FUNCTION_BLOCK "LUps-M"   // FB1313, FBD
TITLE = LUps-M / LUps-M 2012-05-11
{ S7_Optimized_Access := 'FALSE' }
AUTHOR : VCC_JS
FAMILY : Actuator
NAME : LUps
VERSION : 0.2
// ================================================================================
// This module handles alarms from the UPS of type Murr electronic.
// When the conditions to generate the alarm disappear, a boolean output is 
// available to inform the upper level that the alarm can be reset.
// ================================================================================
// stored: AutoNumber false, IsIECCheckEnabled false, SetENOAutomatically False, UDAEnableTagReadback false
   VAR_INPUT
      I_UPSOk { ExternalAccessible := 'False'; ExternalVisible := 'False'; ExternalWritable := 'False'} : Bool;   // Input signal of UPS OK-signal
      I_SupplyVoltageOk { ExternalAccessible := 'False'; ExternalVisible := 'False'; ExternalWritable := 'False'} : Bool;   // Input signal supply voltage OK
      I_CapacitorOk { ExternalAccessible := 'False'; ExternalVisible := 'False'; ExternalWritable := 'False'} : Bool;   // Input signal Capacitor OK
      I_EnableAlarm { ExternalAccessible := 'False'; ExternalVisible := 'False'; ExternalWritable := 'False'} : Bool := TRUE;   // Enable alarm from upper level (0=disable/1=enable)
      I_AlarmResetPB { ExternalAccessible := 'False'; ExternalVisible := 'False'; ExternalWritable := 'False'} : Bool;   // Alarm reset pushbutton is activated
   END_VAR
   VAR_OUTPUT
      O_UPSOk { ExternalAccessible := 'False'; ExternalVisible := 'False'; ExternalWritable := 'False'} : Bool;   // UPS ok
      O_AlarmA { ExternalAccessible := 'False'; ExternalVisible := 'False'; ExternalWritable := 'False'} : Bool;   // Summation Alarm A.
      O_AlarmB { ExternalAccessible := 'False'; ExternalVisible := 'False'; ExternalWritable := 'False'} : Bool;   // Summation Alarm B.
      O_AlarmC { ExternalAccessible := 'False'; ExternalVisible := 'False'; ExternalWritable := 'False'} : Bool;   // Summation Alarm C.
      O_AlarmD { ExternalAccessible := 'False'; ExternalVisible := 'False'; ExternalWritable := 'False'} : Bool;   // Summation Alarm D.
      O_AlarmABCondition { ExternalAccessible := 'False'; ExternalVisible := 'False'; ExternalWritable := 'False'} : Bool;   // Alarm AB Condition
      H_IAnim { ExternalAccessible := 'False'; ExternalVisible := 'False'; ExternalWritable := 'False'} : Word;   // Icon animation
      H_AlarmWord { ExternalAccessible := 'False'; ExternalVisible := 'False'; ExternalWritable := 'False'} : DWord;   // Alarm Word
   END_VAR
   VAR DB_SPECIFIC
      AA_UPSFault { ExternalAccessible := 'False'; ExternalVisible := 'False'; ExternalWritable := 'False'} : Bool;   // UPS Fault / 0000: UPS Fault
      AD_SupplyVoltageAlarm { ExternalAccessible := 'False'; ExternalVisible := 'False'; ExternalWritable := 'False'} : Bool;   // Supply voltage not Ok / 0000: Supply voltage not Ok
      AD_UPSCapacitor { ExternalAccessible := 'False'; ExternalVisible := 'False'; ExternalWritable := 'False'} : Bool;   // UPS Capacitor warning / 0000: UPS Capacitor warning
      H_Out : Struct   // HMI
         Anim : Word;   // HMI Animation of the object
         DBnr : Int;   // HMI Animation DB number
      END_STRUCT;
      UPSCond { ExternalAccessible := 'False'; ExternalVisible := 'False'; ExternalWritable := 'False'} : Bool;   // Input condition to set the UPS alarm
      AlarmA { ExternalAccessible := 'False'; ExternalVisible := 'False'; ExternalWritable := 'False'} : Bool;   // Summation Alarm A
      AlarmB { ExternalAccessible := 'False'; ExternalVisible := 'False'; ExternalWritable := 'False'} : Bool;   // Summation Alarm B
      AlarmC { ExternalAccessible := 'False'; ExternalVisible := 'False'; ExternalWritable := 'False'} : Bool;   // Summation Alarm C
      AlarmD { ExternalAccessible := 'False'; ExternalVisible := 'False'; ExternalWritable := 'False'} : Bool;   // Summation Alarm D
      UPSOk { ExternalAccessible := 'False'; ExternalVisible := 'False'; ExternalWritable := 'False'} : Bool;   // UPS is ok
      DBnr { ExternalAccessible := 'False'; ExternalVisible := 'False'; ExternalWritable := 'False'} : Int;   // DB number
   END_VAR
BEGIN

NETWORK
TITLE = **** 1 - Inputs **** DB number
// DB number
      L     DINO;
      T     #DBnr;

REGION Network 2: **** 1 - Inputs **** The UPS alarm is active / **** 1 - Inputs ****
   // The UPS alarm is active
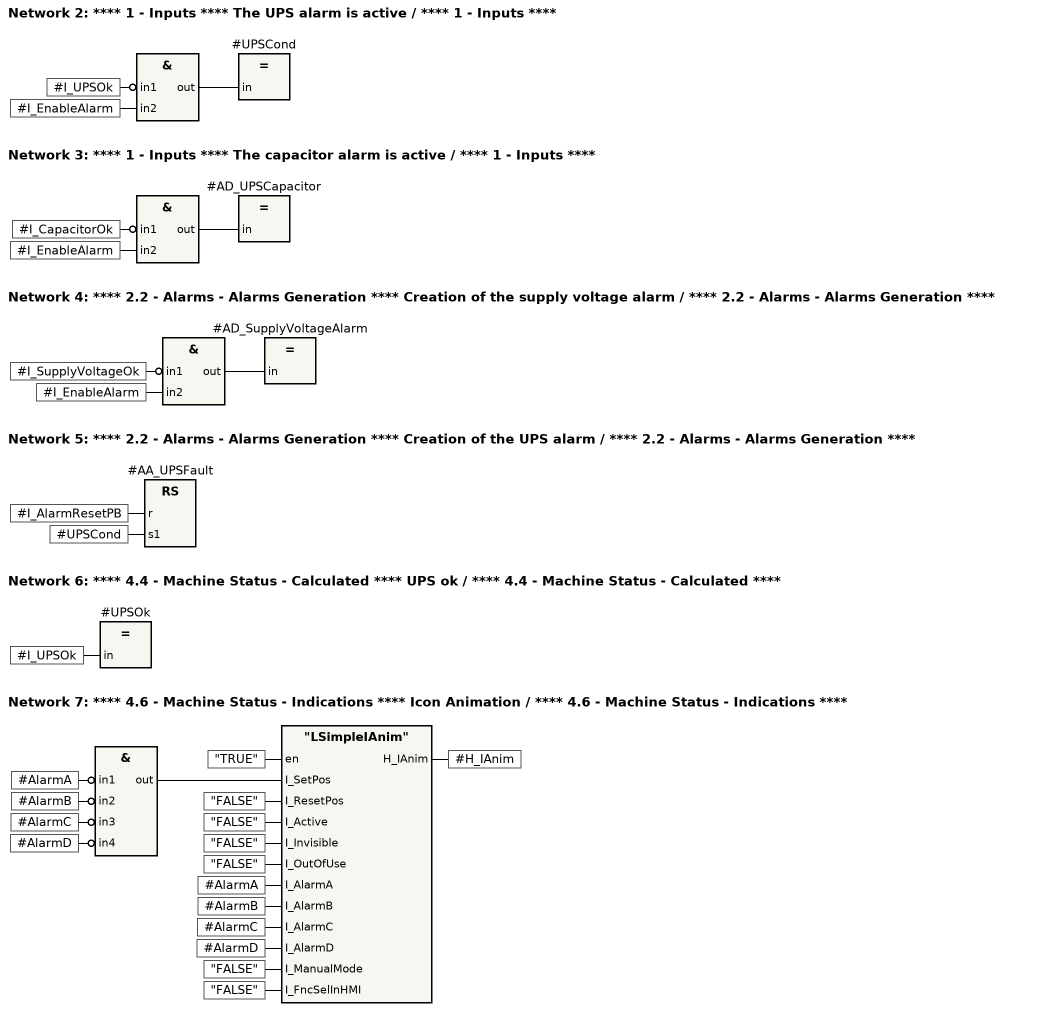
   #UPSCond := NOT #I_UPSOk AND #I_EnableAlarm;
END_REGION

REGION Network 3: **** 1 - Inputs **** The capacitor alarm is active / **** 1 - Inputs ****
   // The capacitor alarm is active
   #AD_UPSCapacitor := NOT #I_CapacitorOk AND #I_EnableAlarm;
END_REGION

REGION Network 4: **** 2.2 - Alarms - Alarms Generation **** Creation of the supply voltage alarm / **** 2.2 - Alarms - Alarms Generation ****
   // Creation of the supply voltage alarm
   #AD_SupplyVoltageAlarm := NOT #I_SupplyVoltageOk AND #I_EnableAlarm;
END_REGION

REGION Network 5: **** 2.2 - Alarms - Alarms Generation **** Creation of the UPS alarm / **** 2.2 - Alarms - Alarms Generation ****
   // Creation of the UPS alarm
   IF #I_AlarmResetPB THEN
       #AA_UPSFault := FALSE;   // RS flip-flop
   END_IF;
   IF #UPSCond THEN #AA_UPSFault := TRUE; END_IF;
END_REGION

REGION Network 6: **** 4.4 - Machine Status - Calculated **** UPS ok / **** 4.4 - Machine Status - Calculated ****
   // UPS ok
   #UPSOk := #I_UPSOk;
END_REGION

REGION Network 7: **** 4.6 - Machine Status - Indications **** Icon Animation / **** 4.6 - Machine Status - Indications ****
   // Icon Animation
   IF "TRUE" THEN
       "LSimpleIAnim"(I_SetPos := NOT #AlarmA AND NOT #AlarmB AND NOT #AlarmC AND NOT #AlarmD,
                      I_ResetPos := "FALSE",
                      I_Active := "FALSE",
                      I_Invisible := "FALSE",
                      I_OutOfUse := "FALSE",
                      I_AlarmA := #AlarmA,
                      I_AlarmB := #AlarmB,
                      I_AlarmC := #AlarmC,
                      I_AlarmD := #AlarmD,
                      I_ManualMode := "FALSE",
                      I_FncSelInHMI := "FALSE",
                      H_IAnim => #H_IAnim);
   END_IF;
END_REGION

REGION Network 8: **** 4.6 - Machine Status - Indications **** Animation / **** 4.6 - Machine Status - Indications ****
   // Animation
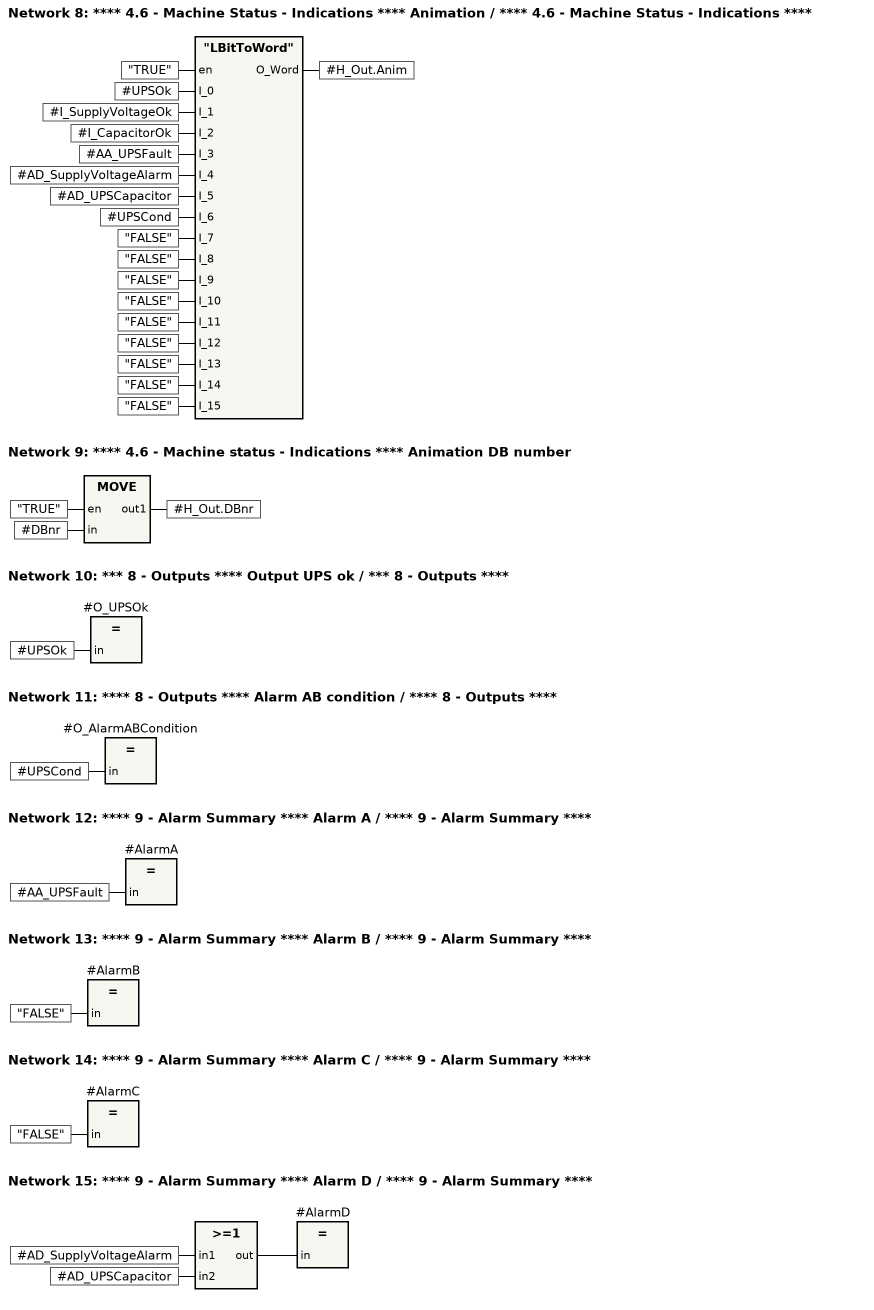
   IF "TRUE" THEN
       "LBitToWord"(I_0 := #UPSOk,
                    I_1 := #I_SupplyVoltageOk,
                    I_2 := #I_CapacitorOk,
                    I_3 := #AA_UPSFault,
                    I_4 := #AD_SupplyVoltageAlarm,
                    I_5 := #AD_UPSCapacitor,
                    I_6 := #UPSCond,
                    I_7 := "FALSE",
                    I_8 := "FALSE",
                    I_9 := "FALSE",
                    I_10 := "FALSE",
                    I_11 := "FALSE",
                    I_12 := "FALSE",
                    I_13 := "FALSE",
                    I_14 := "FALSE",
                    I_15 := "FALSE",
                    O_Word => #H_Out.Anim);
   END_IF;
END_REGION

REGION Network 9: **** 4.6 - Machine status - Indications **** Animation DB number
   // Animation DB number
   IF "TRUE" THEN #H_Out.DBnr := #DBnr; END_IF;
END_REGION

REGION Network 10: *** 8 - Outputs **** Output UPS ok / *** 8 - Outputs ****
   // Output UPS ok
   #O_UPSOk := #UPSOk;
END_REGION

REGION Network 11: **** 8 - Outputs **** Alarm AB condition / **** 8 - Outputs ****
   // Alarm AB Condition
   #O_AlarmABCondition := #UPSCond;
END_REGION

REGION Network 12: **** 9 - Alarm Summary **** Alarm A / **** 9 - Alarm Summary ****
   // Summary of alarms A
   #AlarmA := #AA_UPSFault;
END_REGION

REGION Network 13: **** 9 - Alarm Summary **** Alarm B / **** 9 - Alarm Summary ****
   // Summary of alarms B
   #AlarmB := "FALSE";
END_REGION

REGION Network 14: **** 9 - Alarm Summary **** Alarm C / **** 9 - Alarm Summary ****
   // Summary of alarms C
   #AlarmC := "FALSE";
END_REGION

REGION Network 15: **** 9 - Alarm Summary **** Alarm D / **** 9 - Alarm Summary ****
   // Summary of alarms D
   #AlarmD := #AD_SupplyVoltageAlarm OR #AD_UPSCapacitor;
END_REGION

REGION Network 16: **** 9.1 - Alarm Output **** Alarm A / **** 9 - Alarm Summary ****
   // Output of alarms A
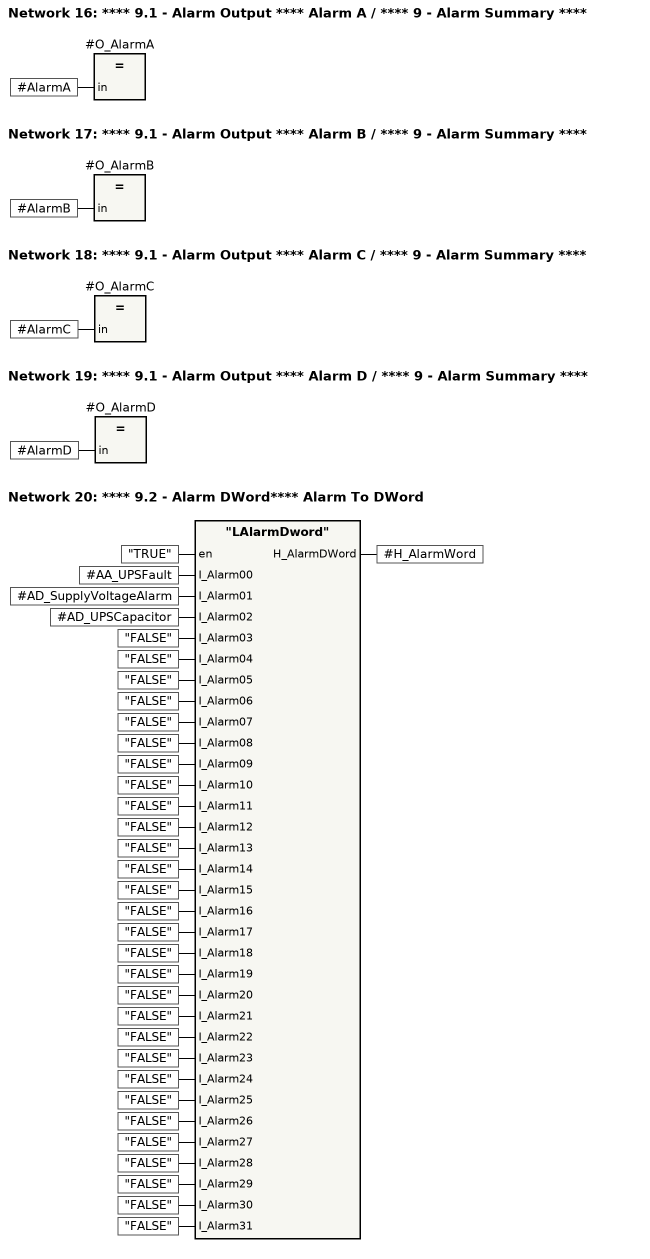
   #O_AlarmA := #AlarmA;
END_REGION

REGION Network 17: **** 9.1 - Alarm Output **** Alarm B / **** 9 - Alarm Summary ****
   // Output of alarms B
   #O_AlarmB := #AlarmB;
END_REGION

REGION Network 18: **** 9.1 - Alarm Output **** Alarm C / **** 9 - Alarm Summary ****
   // Output of alarms C
   #O_AlarmC := #AlarmC;
END_REGION

REGION Network 19: **** 9.1 - Alarm Output **** Alarm D / **** 9 - Alarm Summary ****
   // Output of alarms D
   #O_AlarmD := #AlarmD;
END_REGION

REGION Network 20: **** 9.2 - Alarm DWord**** Alarm To DWord
   // Alarm Word
   IF "TRUE" THEN
       "LAlarmDword"(I_Alarm00 := #AA_UPSFault,
                     I_Alarm01 := #AD_SupplyVoltageAlarm,
                     I_Alarm02 := #AD_UPSCapacitor,
                     I_Alarm03 := "FALSE",
                     I_Alarm04 := "FALSE",
                     I_Alarm05 := "FALSE",
                     I_Alarm06 := "FALSE",
                     I_Alarm07 := "FALSE",
                     I_Alarm08 := "FALSE",
                     I_Alarm09 := "FALSE",
                     I_Alarm10 := "FALSE",
                     I_Alarm11 := "FALSE",
                     I_Alarm12 := "FALSE",
                     I_Alarm13 := "FALSE",
                     I_Alarm14 := "FALSE",
                     I_Alarm15 := "FALSE",
                     I_Alarm16 := "FALSE",
                     I_Alarm17 := "FALSE",
                     I_Alarm18 := "FALSE",
                     I_Alarm19 := "FALSE",
                     I_Alarm20 := "FALSE",
                     I_Alarm21 := "FALSE",
                     I_Alarm22 := "FALSE",
                     I_Alarm23 := "FALSE",
                     I_Alarm24 := "FALSE",
                     I_Alarm25 := "FALSE",
                     I_Alarm26 := "FALSE",
                     I_Alarm27 := "FALSE",
                     I_Alarm28 := "FALSE",
                     I_Alarm29 := "FALSE",
                     I_Alarm30 := "FALSE",
                     I_Alarm31 := "FALSE",
                     H_AlarmDWord => #H_AlarmWord);
   END_IF;
END_REGION
END_FUNCTION_BLOCK

FUNCTION_BLOCK "LUps-Puls"   // FB1314, FBD
TITLE = LUps-M / LUps-M 2012-05-11 / LUps-Puls 2020-07-17
{ S7_Optimized_Access := 'FALSE' }
AUTHOR : VCC_JS
FAMILY : Actuator
NAME : LUps
VERSION : 0.2
// ================================================================================
// This module handles alarms from the UPS of type Murr electronic.
// When the conditions to generate the alarm disappear, a boolean output is 
// available to inform the upper level that the alarm can be reset.
// ================================================================================
// stored: AutoNumber false, IsIECCheckEnabled false, SetENOAutomatically False, UDAEnableTagReadback false
   VAR_INPUT
      I_Active { ExternalAccessible := 'False'; ExternalVisible := 'False'; ExternalWritable := 'False'} : Bool;   // Input signal of UPS Active-Signal / Input signal of UPS OK-signal
      I_Ready { ExternalAccessible := 'False'; ExternalVisible := 'False'; ExternalWritable := 'False'} : Bool;   // Input signal UPS Ready-Signal / Input signal supply voltage OK
      I_EnableAlarm { ExternalAccessible := 'False'; ExternalVisible := 'False'; ExternalWritable := 'False'} : Bool := TRUE;   // Enable alarm from upper level (0=disable/1=enable)
      I_AlarmResetPB { ExternalAccessible := 'False'; ExternalVisible := 'False'; ExternalWritable := 'False'} : Bool;   // Alarm reset pushbutton is activated
   END_VAR
   VAR_OUTPUT
      O_Active { ExternalAccessible := 'False'; ExternalVisible := 'False'; ExternalWritable := 'False'} : Bool;   // UPS Active / UPS ok
      O_AlarmA { ExternalAccessible := 'False'; ExternalVisible := 'False'; ExternalWritable := 'False'} : Bool;   // Summation Alarm A.
      O_AlarmB { ExternalAccessible := 'False'; ExternalVisible := 'False'; ExternalWritable := 'False'} : Bool;   // Summation Alarm B.
      O_AlarmC { ExternalAccessible := 'False'; ExternalVisible := 'False'; ExternalWritable := 'False'} : Bool;   // Summation Alarm C.
      O_AlarmD { ExternalAccessible := 'False'; ExternalVisible := 'False'; ExternalWritable := 'False'} : Bool;   // Summation Alarm D.
      O_AlarmABCondition { ExternalAccessible := 'False'; ExternalVisible := 'False'; ExternalWritable := 'False'} : Bool;   // Alarm AB Condition
      H_IAnim { ExternalAccessible := 'False'; ExternalVisible := 'False'; ExternalWritable := 'False'} : DWord;   // Icon animation
      H_AlarmWord { ExternalAccessible := 'False'; ExternalVisible := 'False'; ExternalWritable := 'False'} : DWord;   // Alarm Word
   END_VAR
   VAR DB_SPECIFIC
      AA_Active { ExternalAccessible := 'False'; ExternalVisible := 'False'; ExternalWritable := 'False'} : Bool;   // UPS Capaciter discharged / UPS Fault / 0000: UPS Fault
      AD_Ready { ExternalAccessible := 'False'; ExternalVisible := 'False'; ExternalWritable := 'False'} : Bool;   // UPS Ready-Signal / Supply voltage not Ok / 0000: Supply voltage not Ok
      H_Out : Struct   // HMI
         Anim : Word;   // HMI Animation of the object
         DBnr : Int;   // HMI Animation DB number
      END_STRUCT;
      UPSActiveAlarmCond { ExternalAccessible := 'False'; ExternalVisible := 'False'; ExternalWritable := 'False'} : Bool;   // Active condition to set the UPS alarm / Input condition to set the UPS alarm
      AlarmA { ExternalAccessible := 'False'; ExternalVisible := 'False'; ExternalWritable := 'False'} : Bool;   // Summation Alarm A
      AlarmB { ExternalAccessible := 'False'; ExternalVisible := 'False'; ExternalWritable := 'False'} : Bool;   // Summation Alarm B
      AlarmC { ExternalAccessible := 'False'; ExternalVisible := 'False'; ExternalWritable := 'False'} : Bool;   // Summation Alarm C
      AlarmD { ExternalAccessible := 'False'; ExternalVisible := 'False'; ExternalWritable := 'False'} : Bool;   // Summation Alarm D
      DBnr { ExternalAccessible := 'False'; ExternalVisible := 'False'; ExternalWritable := 'False'} : Int;   // DB number
   END_VAR
BEGIN

NETWORK
TITLE = **** 1 - Inputs **** DB number
// DB number
      L     DINO;
      T     #DBnr;

REGION Network 2: **** 1 - Inputs **** The UPS alarm is active / **** 1 - Inputs **** / **** 2.2 - Alarms - Alarms Generation **** UPS Not Active alarm condition
   // The UPS alarm is active / UPS Active alarm condition (Capacitors are  being discharged)
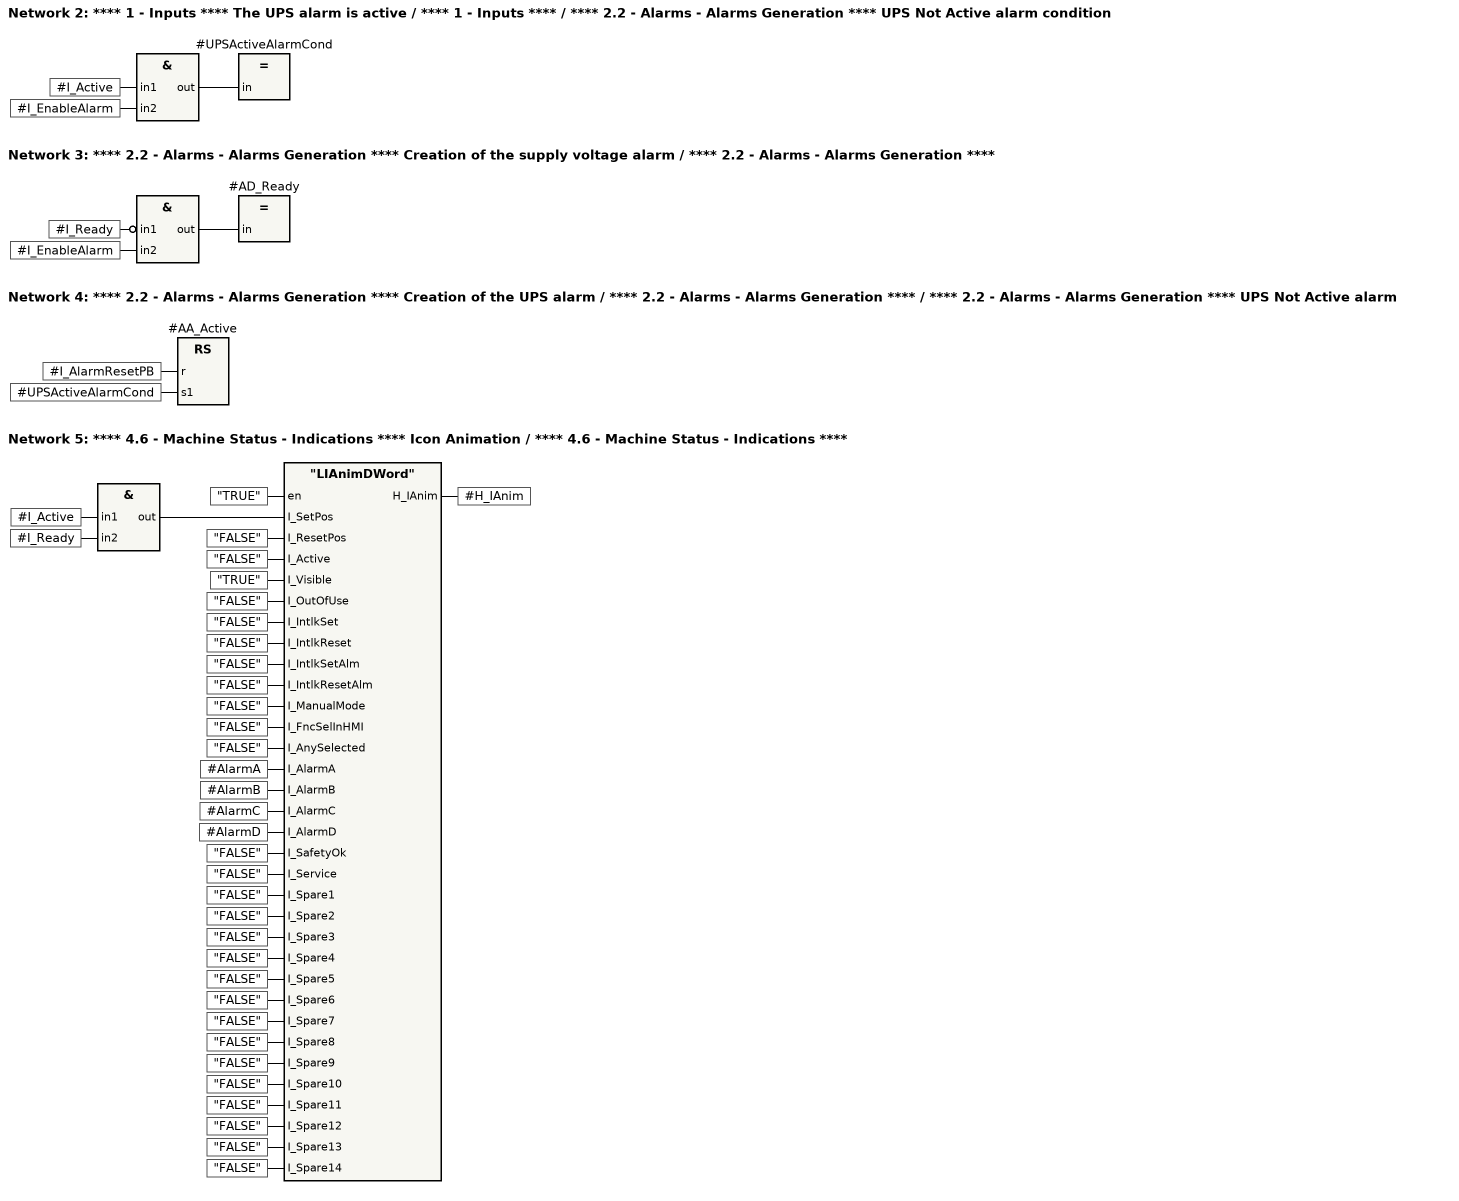
   #UPSActiveAlarmCond := #I_Active AND #I_EnableAlarm;
END_REGION

REGION Network 3: **** 2.2 - Alarms - Alarms Generation **** Creation of the supply voltage alarm / **** 2.2 - Alarms - Alarms Generation ****
   // Creation of the supply voltage alarm
   #AD_Ready := NOT #I_Ready AND #I_EnableAlarm;
END_REGION

REGION Network 4: **** 2.2 - Alarms - Alarms Generation **** Creation of the UPS alarm / **** 2.2 - Alarms - Alarms Generation **** / **** 2.2 - Alarms - Alarms Generation **** UPS Not Active alarm
   // Creation of the UPS alarm
   IF #I_AlarmResetPB THEN
       #AA_Active := FALSE;   // RS flip-flop
   END_IF;
   IF #UPSActiveAlarmCond THEN #AA_Active := TRUE; END_IF;
END_REGION

REGION Network 5: **** 4.6 - Machine Status - Indications **** Icon Animation / **** 4.6 - Machine Status - Indications ****
   // Icon Animation
   IF "TRUE" THEN
       "LIAnimDWord"(I_SetPos := #I_Active AND #I_Ready,
                     I_ResetPos := "FALSE",
                     I_Active := "FALSE",
                     I_Visible := "TRUE",
                     I_OutOfUse := "FALSE",
                     I_IntlkSet := "FALSE",
                     I_IntlkReset := "FALSE",
                     I_IntlkSetAlm := "FALSE",
                     I_IntlkResetAlm := "FALSE",
                     I_ManualMode := "FALSE",
                     I_FncSelInHMI := "FALSE",
                     I_AnySelected := "FALSE",
                     I_AlarmA := #AlarmA,
                     I_AlarmB := #AlarmB,
                     I_AlarmC := #AlarmC,
                     I_AlarmD := #AlarmD,
                     I_SafetyOk := "FALSE",
                     I_Service := "FALSE",
                     I_Spare1 := "FALSE",
                     I_Spare2 := "FALSE",
                     I_Spare3 := "FALSE",
                     I_Spare4 := "FALSE",
                     I_Spare5 := "FALSE",
                     I_Spare6 := "FALSE",
                     I_Spare7 := "FALSE",
                     I_Spare8 := "FALSE",
                     I_Spare9 := "FALSE",
                     I_Spare10 := "FALSE",
                     I_Spare11 := "FALSE",
                     I_Spare12 := "FALSE",
                     I_Spare13 := "FALSE",
                     I_Spare14 := "FALSE",
                     H_IAnim => #H_IAnim);
   END_IF;
END_REGION

REGION Network 6: **** 4.6 - Machine Status - Indications **** Animation / **** 4.6 - Machine Status - Indications ****
   // Animation
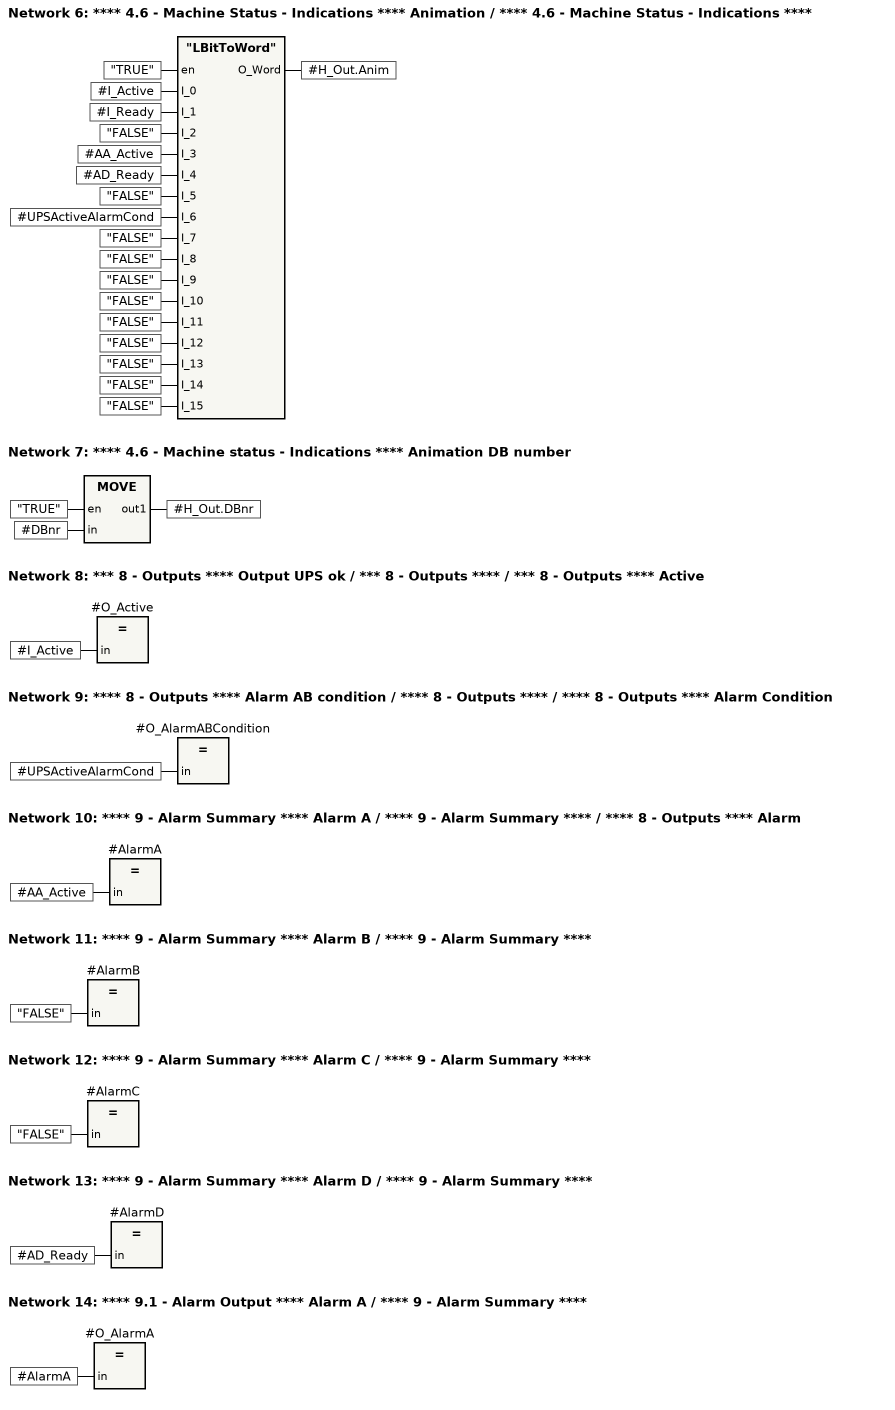
   IF "TRUE" THEN
       "LBitToWord"(I_0 := #I_Active,
                    I_1 := #I_Ready,
                    I_2 := "FALSE",
                    I_3 := #AA_Active,
                    I_4 := #AD_Ready,
                    I_5 := "FALSE",
                    I_6 := #UPSActiveAlarmCond,
                    I_7 := "FALSE",
                    I_8 := "FALSE",
                    I_9 := "FALSE",
                    I_10 := "FALSE",
                    I_11 := "FALSE",
                    I_12 := "FALSE",
                    I_13 := "FALSE",
                    I_14 := "FALSE",
                    I_15 := "FALSE",
                    O_Word => #H_Out.Anim);
   END_IF;
END_REGION

REGION Network 7: **** 4.6 - Machine status - Indications **** Animation DB number
   // Animation DB number
   IF "TRUE" THEN #H_Out.DBnr := #DBnr; END_IF;
END_REGION

REGION Network 8: *** 8 - Outputs **** Output UPS ok / *** 8 - Outputs **** / *** 8 - Outputs **** Active
   // Output UPS ok
   #O_Active := #I_Active;
END_REGION

REGION Network 9: **** 8 - Outputs **** Alarm AB condition / **** 8 - Outputs **** / **** 8 - Outputs **** Alarm Condition
   // Alarm AB Condition
   #O_AlarmABCondition := #UPSActiveAlarmCond;
END_REGION

REGION Network 10: **** 9 - Alarm Summary **** Alarm A / **** 9 - Alarm Summary **** / **** 8 - Outputs **** Alarm
   // Summary of alarms A / Alarm
   #AlarmA := #AA_Active;
END_REGION

REGION Network 11: **** 9 - Alarm Summary **** Alarm B / **** 9 - Alarm Summary ****
   // Summary of alarms B
   #AlarmB := "FALSE";
END_REGION

REGION Network 12: **** 9 - Alarm Summary **** Alarm C / **** 9 - Alarm Summary ****
   // Summary of alarms C
   #AlarmC := "FALSE";
END_REGION

REGION Network 13: **** 9 - Alarm Summary **** Alarm D / **** 9 - Alarm Summary ****
   // Summary of alarms D
   #AlarmD := #AD_Ready;
END_REGION

REGION Network 14: **** 9.1 - Alarm Output **** Alarm A / **** 9 - Alarm Summary ****
   // Output of alarms A
   #O_AlarmA := #AlarmA;
END_REGION

REGION Network 15: **** 9.1 - Alarm Output **** Alarm B / **** 9 - Alarm Summary ****
   // Output of alarms B
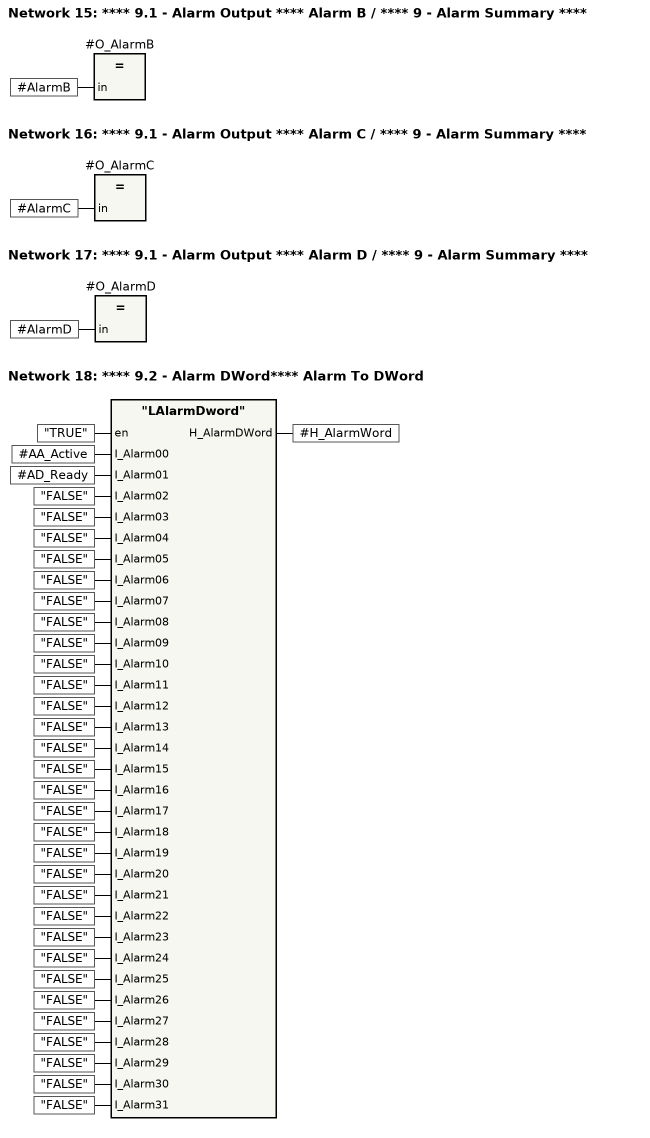
   #O_AlarmB := #AlarmB;
END_REGION

REGION Network 16: **** 9.1 - Alarm Output **** Alarm C / **** 9 - Alarm Summary ****
   // Output of alarms C
   #O_AlarmC := #AlarmC;
END_REGION

REGION Network 17: **** 9.1 - Alarm Output **** Alarm D / **** 9 - Alarm Summary ****
   // Output of alarms D
   #O_AlarmD := #AlarmD;
END_REGION

REGION Network 18: **** 9.2 - Alarm DWord**** Alarm To DWord
   // Alarm Word
   IF "TRUE" THEN
       "LAlarmDword"(I_Alarm00 := #AA_Active,
                     I_Alarm01 := #AD_Ready,
                     I_Alarm02 := "FALSE",
                     I_Alarm03 := "FALSE",
                     I_Alarm04 := "FALSE",
                     I_Alarm05 := "FALSE",
                     I_Alarm06 := "FALSE",
                     I_Alarm07 := "FALSE",
                     I_Alarm08 := "FALSE",
                     I_Alarm09 := "FALSE",
                     I_Alarm10 := "FALSE",
                     I_Alarm11 := "FALSE",
                     I_Alarm12 := "FALSE",
                     I_Alarm13 := "FALSE",
                     I_Alarm14 := "FALSE",
                     I_Alarm15 := "FALSE",
                     I_Alarm16 := "FALSE",
                     I_Alarm17 := "FALSE",
                     I_Alarm18 := "FALSE",
                     I_Alarm19 := "FALSE",
                     I_Alarm20 := "FALSE",
                     I_Alarm21 := "FALSE",
                     I_Alarm22 := "FALSE",
                     I_Alarm23 := "FALSE",
                     I_Alarm24 := "FALSE",
                     I_Alarm25 := "FALSE",
                     I_Alarm26 := "FALSE",
                     I_Alarm27 := "FALSE",
                     I_Alarm28 := "FALSE",
                     I_Alarm29 := "FALSE",
                     I_Alarm30 := "FALSE",
                     I_Alarm31 := "FALSE",
                     H_AlarmDWord => #H_AlarmWord);
   END_IF;
END_REGION
END_FUNCTION_BLOCK

FUNCTION_BLOCK "L1Alarm"   // FB1401, FBD
TITLE = L1Alarm / LProc1Alarm
{ S7_Optimized_Access := 'FALSE' }
AUTHOR : VCC
FAMILY : AlarmHnd
NAME : 1Alarm
VERSION : 1.0
// ================================================================================
// This module is used everywhere one alarm shall be generated when one (security) 
// input becomes True. The alarm have a delay time set in millieseconds.
// The alarm can be True only when the input Enable Alarm is also True.
// 
// When the conditions to generate the alarm is disappear, a boolean output is 
// available to inform the upper level that the alarm can be reset.
// The alarm is reset by means of the AlarmResetPB signal.
// ================================================================================
// stored: AutoNumber false, IsIECCheckEnabled false, SetENOAutomatically False, UDAEnableTagReadback false
   VAR_INPUT
      I_Input { ExternalAccessible := 'False'; ExternalVisible := 'False'; ExternalWritable := 'False'} : Bool;   // Input signal of the alarm
      I_AlarmClass { ExternalAccessible := 'False'; ExternalVisible := 'False'; ExternalWritable := 'False'} : Char;   // Alarm class -> A - B - C - D or E
      I_EnableAlarm { ExternalAccessible := 'False'; ExternalVisible := 'False'; ExternalWritable := 'False'} : Bool := TRUE;   // Enable alarm from upper level
      I_AlarmResetPB { ExternalAccessible := 'False'; ExternalVisible := 'False'; ExternalWritable := 'False'} : Bool;   // Alarm reset pushbutton is activated
      I_Invisible { ExternalAccessible := 'False'; ExternalVisible := 'False'; ExternalWritable := 'False'} : Bool;   // Invisible
      C_NcAlarm { ExternalAccessible := 'False'; ExternalVisible := 'False'; ExternalWritable := 'False'} : Bool;   // Alarm contact NC
   END_VAR
   VAR_OUTPUT
      O_Alarm { ExternalAccessible := 'False'; ExternalVisible := 'False'; ExternalWritable := 'False'} : Bool;   // Alarm
      O_AlarmABCondition { ExternalAccessible := 'False'; ExternalVisible := 'False'; ExternalWritable := 'False'} : Bool;   // Alarm AB condition
      H_IAnim { ExternalAccessible := 'False'; ExternalVisible := 'False'; ExternalWritable := 'False'} : Word;   // Icon animation
   END_VAR
   VAR DB_SPECIFIC
      H_Out : Struct   // HMI
         Anim : Word;   // HMI Animation of the object
         DBnr : Int;   // HMI Animation DB number
      END_STRUCT;
      Alarm { ExternalAccessible := 'False'; ExternalVisible := 'False'; ExternalWritable := 'False'} : Bool;   // Alarm
      AlarmClass_A { ExternalAccessible := 'False'; ExternalVisible := 'False'; ExternalWritable := 'False'} : Bool;   // The alarm is from alarm class A
      AlarmClass_B { ExternalAccessible := 'False'; ExternalVisible := 'False'; ExternalWritable := 'False'} : Bool;   // The alarm is from alarm class B
      AlarmClass_C { ExternalAccessible := 'False'; ExternalVisible := 'False'; ExternalWritable := 'False'} : Bool;   // The alarm is from alarm class C
      AlarmClass_D { ExternalAccessible := 'False'; ExternalVisible := 'False'; ExternalWritable := 'False'} : Bool;   // The alarm is from alarm class D
      AlarmClass_E { ExternalAccessible := 'False'; ExternalVisible := 'False'; ExternalWritable := 'False'} : Bool;   // The alarm is from alarm class E
      AlarmCond { ExternalAccessible := 'False'; ExternalVisible := 'False'; ExternalWritable := 'False'} : Bool;   // Alarm condition
      DBnr { ExternalAccessible := 'False'; ExternalVisible := 'False'; ExternalWritable := 'False'} : Int;   // HMI DB number
   END_VAR
BEGIN

NETWORK
TITLE = **** 1 - Inputs **** DB number
// DB number
      L     DINO;
      T     #DBnr;

NETWORK
TITLE = **** 1 - Inputs **** Alarm class
// Alarm class
// Alarm class = E
      L     #I_AlarmClass;
      L     'E';
      ==I;
      =     #AlarmClass_E;

// Alarm class = D
      L     #I_AlarmClass;
      L     'D';
      ==I;
      =     #AlarmClass_D;

// Alarm class = C
      L     #I_AlarmClass;
      L     'C';
      ==I;
      =     #AlarmClass_C;

// Alarm class = B
      L     #I_AlarmClass;
      L     'B';
      ==I;
      =     #AlarmClass_B;

// Alarm class = A
      AN    #AlarmClass_B;
      AN    #AlarmClass_C;
      AN    #AlarmClass_D;
      AN    #AlarmClass_E;
      =     #AlarmClass_A;


REGION Network 3: **** 2.2 - Alarms - Alarms Generation **** Alarm Condition
   // Condition for the Alarm
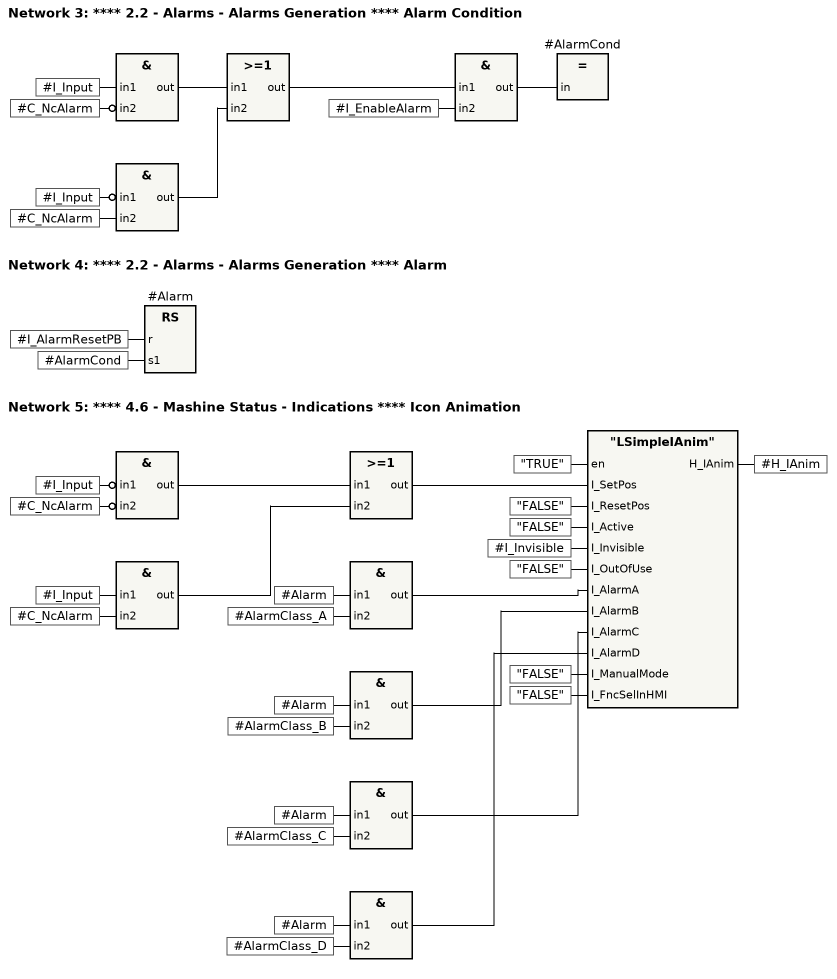
   #AlarmCond := ((#I_Input AND NOT #C_NcAlarm) OR (NOT #I_Input AND #C_NcAlarm)) AND #I_EnableAlarm;
END_REGION

REGION Network 4: **** 2.2 - Alarms - Alarms Generation **** Alarm
   // Creation of the Alarm
   IF #I_AlarmResetPB THEN
       #Alarm := FALSE;   // RS flip-flop
   END_IF;
   IF #AlarmCond THEN #Alarm := TRUE; END_IF;
END_REGION

REGION Network 5: **** 4.6 - Mashine Status - Indications **** Icon Animation
   // Icon Animation
   IF "TRUE" THEN
       "LSimpleIAnim"(I_SetPos := (NOT #I_Input AND NOT #C_NcAlarm) OR (#I_Input AND #C_NcAlarm),
                      I_ResetPos := "FALSE",
                      I_Active := "FALSE",
                      I_Invisible := #I_Invisible,
                      I_OutOfUse := "FALSE",
                      I_AlarmA := #Alarm AND #AlarmClass_A,
                      I_AlarmB := #Alarm AND #AlarmClass_B,
                      I_AlarmC := #Alarm AND #AlarmClass_C,
                      I_AlarmD := #Alarm AND #AlarmClass_D,
                      I_ManualMode := "FALSE",
                      I_FncSelInHMI := "FALSE",
                      H_IAnim => #H_IAnim);
   END_IF;
END_REGION

REGION Network 6: **** 4.6 - Machine Status - Indications **** Animation
   // Animation
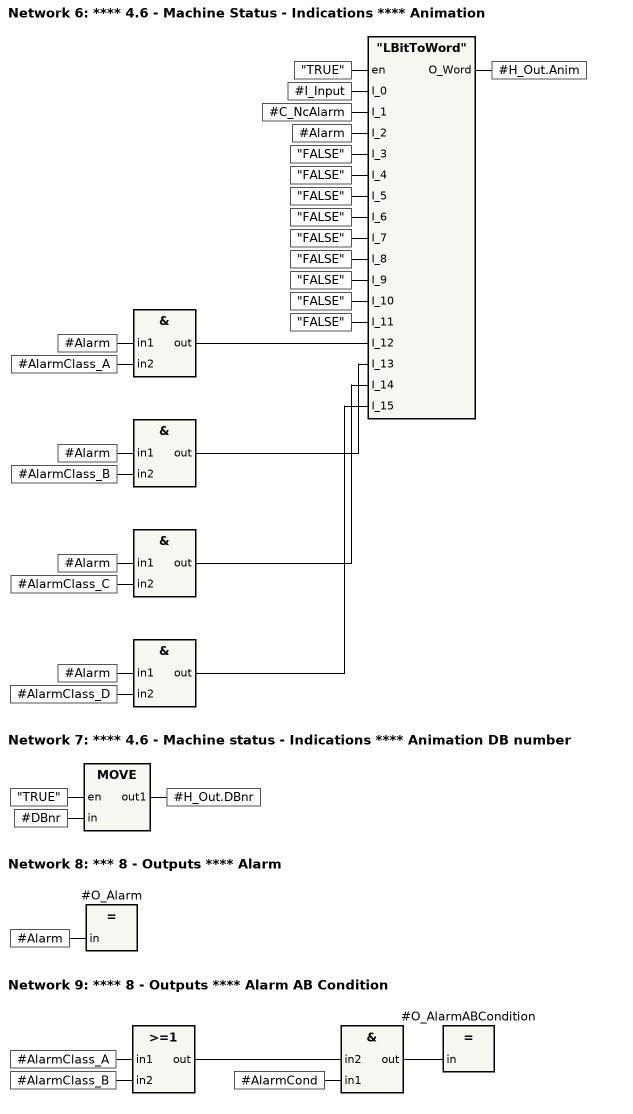
   IF "TRUE" THEN
       "LBitToWord"(I_0 := #I_Input,
                    I_1 := #C_NcAlarm,
                    I_2 := #Alarm,
                    I_3 := "FALSE",
                    I_4 := "FALSE",
                    I_5 := "FALSE",
                    I_6 := "FALSE",
                    I_7 := "FALSE",
                    I_8 := "FALSE",
                    I_9 := "FALSE",
                    I_10 := "FALSE",
                    I_11 := "FALSE",
                    I_12 := #Alarm AND #AlarmClass_A,
                    I_13 := #Alarm AND #AlarmClass_B,
                    I_14 := #Alarm AND #AlarmClass_C,
                    I_15 := #Alarm AND #AlarmClass_D,
                    O_Word => #H_Out.Anim);
   END_IF;
END_REGION

REGION Network 7: **** 4.6 - Machine status - Indications **** Animation DB number
   // Animation DB number
   IF "TRUE" THEN #H_Out.DBnr := #DBnr; END_IF;
END_REGION

REGION Network 8: *** 8 - Outputs **** Alarm
   // Output of the Alarm
   #O_Alarm := #Alarm;
END_REGION

REGION Network 9: **** 8 - Outputs **** Alarm AB Condition
   // Alarm Resetable
   #O_AlarmABCondition := (#AlarmClass_A OR #AlarmClass_B) AND #AlarmCond;
END_REGION
END_FUNCTION_BLOCK

FUNCTION_BLOCK "L5Alarm"   // FB1405, FBD
TITLE = L5Alarm
{ S7_Optimized_Access := 'FALSE' }
AUTHOR : VCC
FAMILY : AlarmHnd
NAME : 5Alarm
VERSION : 1.0
// ================================================================================
// This module is used everywhere 5 alarms has to be generated when one (security) 
// corresponding input becomes True.
// All alarms can be True only when the corresponding input Enable Alarm is also 
// True.
// When the conditions to generate the alarm is disappear, a boolean (one per 
// alarm) available to inform the upper level that the corresponding alarm can be 
// reset.
// All alarms are reset by means of the AlarmResetPB signal.
// ================================================================================
// stored: AutoNumber false, IsIECCheckEnabled false, SetENOAutomatically False, UDAEnableTagReadback false
   VAR_INPUT
      I_Input1 { ExternalAccessible := 'False'; ExternalVisible := 'False'; ExternalWritable := 'False'} : Bool;   // Input alarm 1
      I_AlarmClass1 { ExternalAccessible := 'False'; ExternalVisible := 'False'; ExternalWritable := 'False'} : Char;   // Alarm class -> A - B - C - D or E
      I_EnableAlarm1 { ExternalAccessible := 'False'; ExternalVisible := 'False'; ExternalWritable := 'False'} : Bool := TRUE;   // Enable alarm 1 from upper level
      I_Invisible1 { ExternalAccessible := 'False'; ExternalVisible := 'False'; ExternalWritable := 'False'} : Bool;   // Invisible 1
      I_Input2 { ExternalAccessible := 'False'; ExternalVisible := 'False'; ExternalWritable := 'False'} : Bool;   // Input alarm 2
      I_AlarmClass2 { ExternalAccessible := 'False'; ExternalVisible := 'False'; ExternalWritable := 'False'} : Char;   // Alarm class -> A - B - C - D or E
      I_EnableAlarm2 { ExternalAccessible := 'False'; ExternalVisible := 'False'; ExternalWritable := 'False'} : Bool := TRUE;   // Enable alarm 2 from upper level
      I_Invisible2 { ExternalAccessible := 'False'; ExternalVisible := 'False'; ExternalWritable := 'False'} : Bool;   // Invisible 2
      I_Input3 { ExternalAccessible := 'False'; ExternalVisible := 'False'; ExternalWritable := 'False'} : Bool;   // Input alarm 3
      I_AlarmClass3 { ExternalAccessible := 'False'; ExternalVisible := 'False'; ExternalWritable := 'False'} : Char;   // Alarm class -> A - B - C - D or E
      I_EnableAlarm3 { ExternalAccessible := 'False'; ExternalVisible := 'False'; ExternalWritable := 'False'} : Bool := TRUE;   // Enable alarm 3 from upper level
      I_Invisible3 { ExternalAccessible := 'False'; ExternalVisible := 'False'; ExternalWritable := 'False'} : Bool;   // Invisible 3
      I_Input4 { ExternalAccessible := 'False'; ExternalVisible := 'False'; ExternalWritable := 'False'} : Bool;   // Input alarm 4
      I_AlarmClass4 { ExternalAccessible := 'False'; ExternalVisible := 'False'; ExternalWritable := 'False'} : Char;   // Alarm class -> A - B - C - D or E
      I_EnableAlarm4 { ExternalAccessible := 'False'; ExternalVisible := 'False'; ExternalWritable := 'False'} : Bool := TRUE;   // Enable alarm 4 from upper level
      I_Invisible4 { ExternalAccessible := 'False'; ExternalVisible := 'False'; ExternalWritable := 'False'} : Bool;   // Invisible 4
      I_Input5 { ExternalAccessible := 'False'; ExternalVisible := 'False'; ExternalWritable := 'False'} : Bool;   // Input alarm 5
      I_AlarmClass5 { ExternalAccessible := 'False'; ExternalVisible := 'False'; ExternalWritable := 'False'} : Char;   // Alarm class -> A - B - C - D or E
      I_EnableAlarm5 { ExternalAccessible := 'False'; ExternalVisible := 'False'; ExternalWritable := 'False'} : Bool := TRUE;   // Enable alarm 5 from upper level
      I_Invisible5 { ExternalAccessible := 'False'; ExternalVisible := 'False'; ExternalWritable := 'False'} : Bool;   // Invisible
      I_AlarmResetPB { ExternalAccessible := 'False'; ExternalVisible := 'False'; ExternalWritable := 'False'} : Bool;   // Alarm reset pushbutton is activated
   END_VAR
   VAR_OUTPUT
      O_Alarm1 { ExternalAccessible := 'False'; ExternalVisible := 'False'; ExternalWritable := 'False'} : Bool;   // Alarm 1
      O_Alarm2 { ExternalAccessible := 'False'; ExternalVisible := 'False'; ExternalWritable := 'False'} : Bool;   // Alarm 2
      O_Alarm3 { ExternalAccessible := 'False'; ExternalVisible := 'False'; ExternalWritable := 'False'} : Bool;   // Alarm 3
      O_Alarm4 { ExternalAccessible := 'False'; ExternalVisible := 'False'; ExternalWritable := 'False'} : Bool;   // Alarm 4
      O_Alarm5 { ExternalAccessible := 'False'; ExternalVisible := 'False'; ExternalWritable := 'False'} : Bool;   // Alarm 5
      O_AlarmABCondition { ExternalAccessible := 'False'; ExternalVisible := 'False'; ExternalWritable := 'False'} : Bool;   // Alarm AB condition
      H_IAnim1 { ExternalAccessible := 'False'; ExternalVisible := 'False'; ExternalWritable := 'False'} : Word;   // Icon Animation 1
      H_IAnim2 { ExternalAccessible := 'False'; ExternalVisible := 'False'; ExternalWritable := 'False'} : Word;   // Icon Animation 2
      H_IAnim3 { ExternalAccessible := 'False'; ExternalVisible := 'False'; ExternalWritable := 'False'} : Word;   // Icon Animation 3
      H_IAnim4 { ExternalAccessible := 'False'; ExternalVisible := 'False'; ExternalWritable := 'False'} : Word;   // Icon Animation 4
      H_IAnim5 { ExternalAccessible := 'False'; ExternalVisible := 'False'; ExternalWritable := 'False'} : Word;   // Icon Animation 5
   END_VAR
   VAR DB_SPECIFIC
      H_Out : Struct   // HMI
         Anim1 : Word;   // HMI Animation of the object
         Anim2 : Word;   // HMI Animation of the object
         Anim3 : Word;   // HMI Animation of the object
         Anim4 : Word;   // HMI Animation of the object
         Anim5 : Word;   // HMI Animation of the object
         DBnr : Int;   // HMI Animation DB number
      END_STRUCT;
      Alarm1 { ExternalAccessible := 'False'; ExternalVisible := 'False'; ExternalWritable := 'False'} : Bool;   // Alarm 1
      AlarmClass1_A { ExternalAccessible := 'False'; ExternalVisible := 'False'; ExternalWritable := 'False'} : Bool;   // The alarm is from alarm class A
      AlarmClass1_B { ExternalAccessible := 'False'; ExternalVisible := 'False'; ExternalWritable := 'False'} : Bool;   // The alarm is from alarm class B
      AlarmClass1_C { ExternalAccessible := 'False'; ExternalVisible := 'False'; ExternalWritable := 'False'} : Bool;   // The alarm is from alarm class C
      AlarmClass1_D { ExternalAccessible := 'False'; ExternalVisible := 'False'; ExternalWritable := 'False'} : Bool;   // The alarm is from alarm class D
      AlarmClass1_E { ExternalAccessible := 'False'; ExternalVisible := 'False'; ExternalWritable := 'False'} : Bool;   // The alarm is from alarm class E
      Alarm1Cond { ExternalAccessible := 'False'; ExternalVisible := 'False'; ExternalWritable := 'False'} : Bool;   // Alarm 1 condition
      Alarm2 { ExternalAccessible := 'False'; ExternalVisible := 'False'; ExternalWritable := 'False'} : Bool;   // Alarm 2
      AlarmClass2_A { ExternalAccessible := 'False'; ExternalVisible := 'False'; ExternalWritable := 'False'} : Bool;   // The alarm is from alarm class A
      AlarmClass2_B { ExternalAccessible := 'False'; ExternalVisible := 'False'; ExternalWritable := 'False'} : Bool;   // The alarm is from alarm class B
      AlarmClass2_C { ExternalAccessible := 'False'; ExternalVisible := 'False'; ExternalWritable := 'False'} : Bool;   // The alarm is from alarm class C
      AlarmClass2_D { ExternalAccessible := 'False'; ExternalVisible := 'False'; ExternalWritable := 'False'} : Bool;   // The alarm is from alarm class D
      AlarmClass2_E { ExternalAccessible := 'False'; ExternalVisible := 'False'; ExternalWritable := 'False'} : Bool;   // The alarm is from alarm class E
      Alarm2Cond { ExternalAccessible := 'False'; ExternalVisible := 'False'; ExternalWritable := 'False'} : Bool;   // Alarm 2 condition
      Alarm3 { ExternalAccessible := 'False'; ExternalVisible := 'False'; ExternalWritable := 'False'} : Bool;   // Alarm 3
      AlarmClass3_A { ExternalAccessible := 'False'; ExternalVisible := 'False'; ExternalWritable := 'False'} : Bool;   // The alarm is from alarm class A
      AlarmClass3_B { ExternalAccessible := 'False'; ExternalVisible := 'False'; ExternalWritable := 'False'} : Bool;   // The alarm is from alarm class B
      AlarmClass3_C { ExternalAccessible := 'False'; ExternalVisible := 'False'; ExternalWritable := 'False'} : Bool;   // The alarm is from alarm class C
      AlarmClass3_D { ExternalAccessible := 'False'; ExternalVisible := 'False'; ExternalWritable := 'False'} : Bool;   // The alarm is from alarm class D
      AlarmClass3_E { ExternalAccessible := 'False'; ExternalVisible := 'False'; ExternalWritable := 'False'} : Bool;   // The alarm is from alarm class E
      Alarm3Cond { ExternalAccessible := 'False'; ExternalVisible := 'False'; ExternalWritable := 'False'} : Bool;   // Alarm 3 condition
      Alarm4 { ExternalAccessible := 'False'; ExternalVisible := 'False'; ExternalWritable := 'False'} : Bool;   // Alarm 4
      AlarmClass4_A { ExternalAccessible := 'False'; ExternalVisible := 'False'; ExternalWritable := 'False'} : Bool;   // The alarm is from alarm class A
      AlarmClass4_B { ExternalAccessible := 'False'; ExternalVisible := 'False'; ExternalWritable := 'False'} : Bool;   // The alarm is from alarm class B
      AlarmClass4_C { ExternalAccessible := 'False'; ExternalVisible := 'False'; ExternalWritable := 'False'} : Bool;   // The alarm is from alarm class C
      AlarmClass4_D { ExternalAccessible := 'False'; ExternalVisible := 'False'; ExternalWritable := 'False'} : Bool;   // The alarm is from alarm class D
      AlarmClass4_E { ExternalAccessible := 'False'; ExternalVisible := 'False'; ExternalWritable := 'False'} : Bool;   // The alarm is from alarm class E
      Alarm4Cond { ExternalAccessible := 'False'; ExternalVisible := 'False'; ExternalWritable := 'False'} : Bool;   // Alarm 4 condition
      Alarm5 { ExternalAccessible := 'False'; ExternalVisible := 'False'; ExternalWritable := 'False'} : Bool;   // Alarm 5
      AlarmClass5_A { ExternalAccessible := 'False'; ExternalVisible := 'False'; ExternalWritable := 'False'} : Bool;   // The alarm is from alarm class A
      AlarmClass5_B { ExternalAccessible := 'False'; ExternalVisible := 'False'; ExternalWritable := 'False'} : Bool;   // The alarm is from alarm class B
      AlarmClass5_C { ExternalAccessible := 'False'; ExternalVisible := 'False'; ExternalWritable := 'False'} : Bool;   // The alarm is from alarm class C
      AlarmClass5_D { ExternalAccessible := 'False'; ExternalVisible := 'False'; ExternalWritable := 'False'} : Bool;   // The alarm is from alarm class D
      AlarmClass5_E { ExternalAccessible := 'False'; ExternalVisible := 'False'; ExternalWritable := 'False'} : Bool;   // The alarm is from alarm class E
      Alarm5Cond { ExternalAccessible := 'False'; ExternalVisible := 'False'; ExternalWritable := 'False'} : Bool;   // Alarm 5 condition
      DBnr { ExternalAccessible := 'False'; ExternalVisible := 'False'; ExternalWritable := 'False'} : Int;   // HMI DB number
   END_VAR
BEGIN

NETWORK
TITLE = **** 1 - Inputs **** DB number
// DB number
      L     DINO;
      T     #DBnr;

NETWORK
TITLE = **** 1 - Inputs **** Alarm class 1
// Alarm class
// Alarm class = E
      L     #I_AlarmClass1;
      L     'E';
      ==I;
      =     #AlarmClass1_E;

// Alarm class = D
      L     #I_AlarmClass1;
      L     'D';
      ==I;
      =     #AlarmClass1_D;

// Alarm class = C
      L     #I_AlarmClass1;
      L     'C';
      ==I;
      =     #AlarmClass1_C;

// Alarm class = B
      L     #I_AlarmClass1;
      L     'B';
      ==I;
      =     #AlarmClass1_B;

// Alarm class = A
      AN    #AlarmClass1_B;
      AN    #AlarmClass1_C;
      AN    #AlarmClass1_D;
      AN    #AlarmClass1_E;
      =     #AlarmClass1_A;


NETWORK
TITLE = **** 1 - Inputs **** Alarm class 2
// Alarm class
// Alarm class = E
      L     #I_AlarmClass2;
      L     'E';
      ==I;
      =     #AlarmClass2_E;

// Alarm class = D
      L     #I_AlarmClass2;
      L     'D';
      ==I;
      =     #AlarmClass2_D;

// Alarm class = C
      L     #I_AlarmClass2;
      L     'C';
      ==I;
      =     #AlarmClass2_C;

// Alarm class = B
      L     #I_AlarmClass2;
      L     'B';
      ==I;
      =     #AlarmClass2_B;

// Alarm class = A
      AN    #AlarmClass2_B;
      AN    #AlarmClass2_C;
      AN    #AlarmClass2_D;
      AN    #AlarmClass2_E;
      =     #AlarmClass2_A;


NETWORK
TITLE = **** 1 - Inputs **** Alarm class 3
// Alarm class
// Alarm class = E
      L     #I_AlarmClass3;
      L     'E';
      ==I;
      =     #AlarmClass3_E;

// Alarm class = D
      L     #I_AlarmClass3;
      L     'D';
      ==I;
      =     #AlarmClass3_D;

// Alarm class = C
      L     #I_AlarmClass3;
      L     'C';
      ==I;
      =     #AlarmClass3_C;

// Alarm class = B
      L     #I_AlarmClass3;
      L     'B';
      ==I;
      =     #AlarmClass3_B;

// Alarm class = A
      AN    #AlarmClass3_B;
      AN    #AlarmClass3_C;
      AN    #AlarmClass3_D;
      AN    #AlarmClass3_E;
      =     #AlarmClass3_A;


NETWORK
TITLE = **** 1 - Inputs **** Alarm class 4
// Alarm class
// Alarm class = E
      L     #I_AlarmClass4;
      L     'E';
      ==I;
      =     #AlarmClass4_E;

// Alarm class = D
      L     #I_AlarmClass4;
      L     'D';
      ==I;
      =     #AlarmClass4_D;

// Alarm class = C
      L     #I_AlarmClass4;
      L     'C';
      ==I;
      =     #AlarmClass4_C;

// Alarm class = B
      L     #I_AlarmClass4;
      L     'B';
      ==I;
      =     #AlarmClass4_B;

// Alarm class = A
      AN    #AlarmClass4_B;
      AN    #AlarmClass4_C;
      AN    #AlarmClass4_D;
      AN    #AlarmClass4_E;
      =     #AlarmClass4_A;


NETWORK
TITLE = **** 1 - Inputs **** Alarm class 5
// Alarm class
// Alarm class = E
      L     #I_AlarmClass5;
      L     'E';
      ==I;
      =     #AlarmClass5_E;

// Alarm class = D
      L     #I_AlarmClass5;
      L     'D';
      ==I;
      =     #AlarmClass5_D;

// Alarm class = C
      L     #I_AlarmClass5;
      L     'C';
      ==I;
      =     #AlarmClass5_C;

// Alarm class = B
      L     #I_AlarmClass5;
      L     'B';
      ==I;
      =     #AlarmClass5_B;

// Alarm class = A
      AN    #AlarmClass5_B;
      AN    #AlarmClass5_C;
      AN    #AlarmClass5_D;
      AN    #AlarmClass5_E;
      =     #AlarmClass5_A;


REGION Network 7: **** 2.2 - Alarms - Alarms Generation **** Alarm Condition 1
   // Condition for Alarm 1
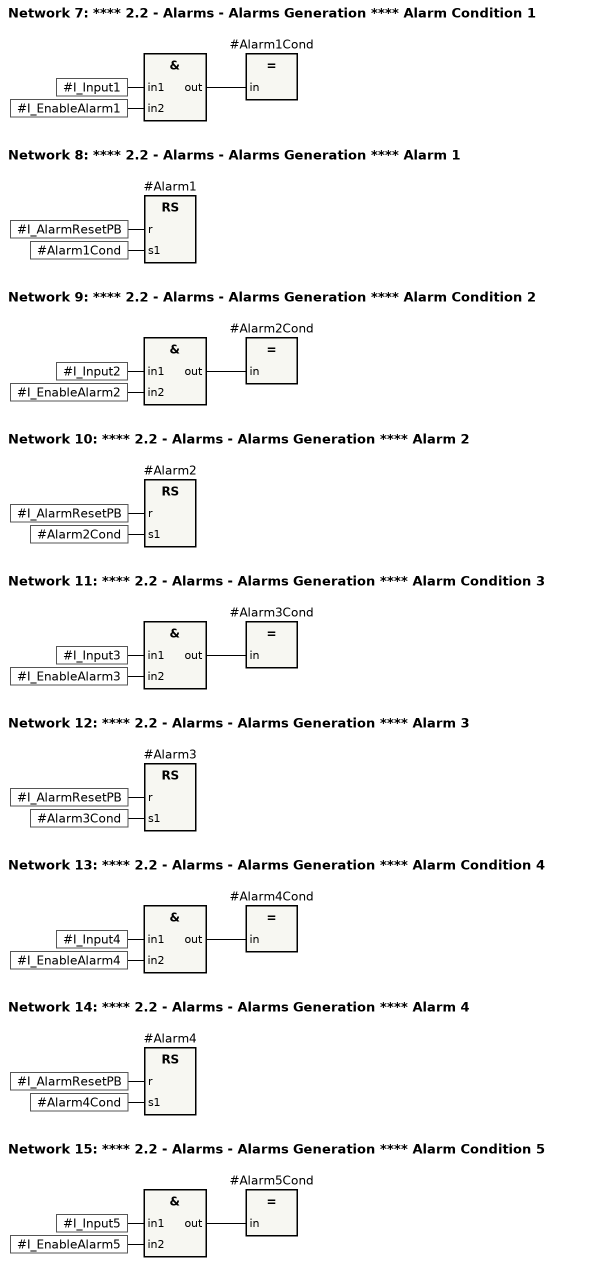
   #Alarm1Cond := #I_Input1 AND #I_EnableAlarm1;
END_REGION

REGION Network 8: **** 2.2 - Alarms - Alarms Generation **** Alarm 1
   // Creation of the Alarm 1
   IF #I_AlarmResetPB THEN
       #Alarm1 := FALSE;   // RS flip-flop
   END_IF;
   IF #Alarm1Cond THEN #Alarm1 := TRUE; END_IF;
END_REGION

REGION Network 9: **** 2.2 - Alarms - Alarms Generation **** Alarm Condition 2
   // Condition for Alarm 2
   #Alarm2Cond := #I_Input2 AND #I_EnableAlarm2;
END_REGION

REGION Network 10: **** 2.2 - Alarms - Alarms Generation **** Alarm 2
   // Creation of the Alarm 2
   IF #I_AlarmResetPB THEN
       #Alarm2 := FALSE;   // RS flip-flop
   END_IF;
   IF #Alarm2Cond THEN #Alarm2 := TRUE; END_IF;
END_REGION

REGION Network 11: **** 2.2 - Alarms - Alarms Generation **** Alarm Condition 3
   // Condition for Alarm 3
   #Alarm3Cond := #I_Input3 AND #I_EnableAlarm3;
END_REGION

REGION Network 12: **** 2.2 - Alarms - Alarms Generation **** Alarm 3
   // Creation of the Alarm 3
   IF #I_AlarmResetPB THEN
       #Alarm3 := FALSE;   // RS flip-flop
   END_IF;
   IF #Alarm3Cond THEN #Alarm3 := TRUE; END_IF;
END_REGION

REGION Network 13: **** 2.2 - Alarms - Alarms Generation **** Alarm Condition 4
   // Condition for Alarm 4
   #Alarm4Cond := #I_Input4 AND #I_EnableAlarm4;
END_REGION

REGION Network 14: **** 2.2 - Alarms - Alarms Generation **** Alarm 4
   // Creation of the Alarm 4
   IF #I_AlarmResetPB THEN
       #Alarm4 := FALSE;   // RS flip-flop
   END_IF;
   IF #Alarm4Cond THEN #Alarm4 := TRUE; END_IF;
END_REGION

REGION Network 15: **** 2.2 - Alarms - Alarms Generation **** Alarm Condition 5
   // Condition for Alarm 5
   #Alarm5Cond := #I_Input5 AND #I_EnableAlarm5;
END_REGION

REGION Network 16: **** 2.2 - Alarms - Alarms Generation **** Alarm 5
   // Creation of the Alarm 5
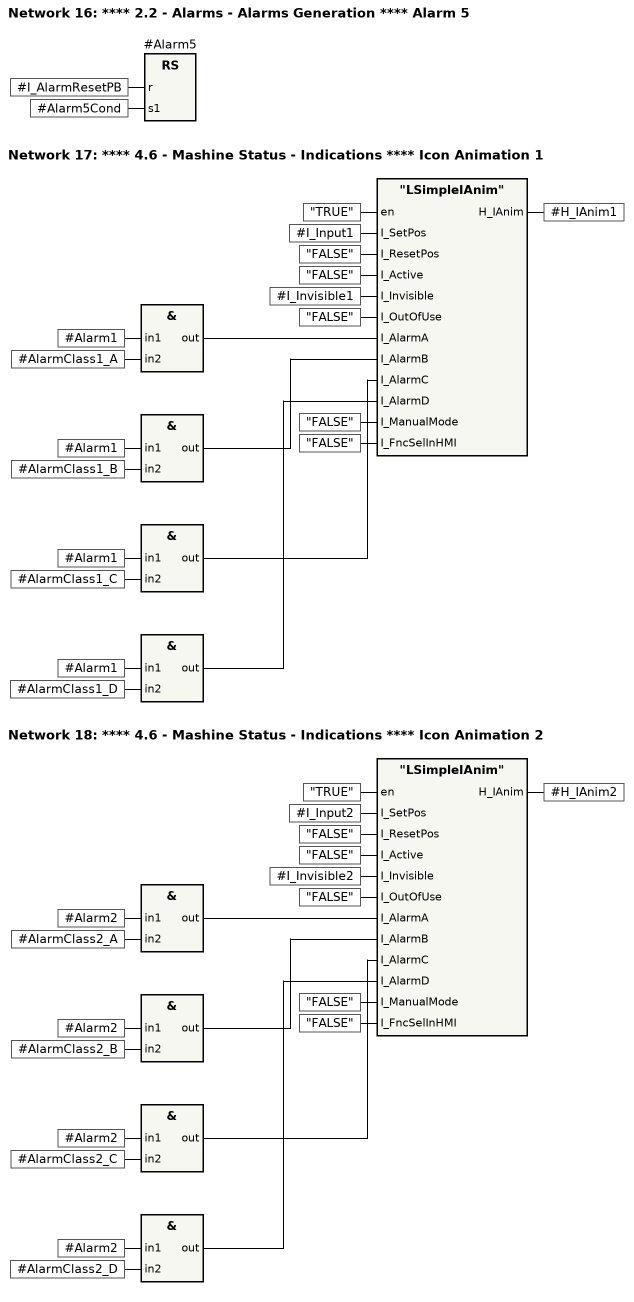
   IF #I_AlarmResetPB THEN
       #Alarm5 := FALSE;   // RS flip-flop
   END_IF;
   IF #Alarm5Cond THEN #Alarm5 := TRUE; END_IF;
END_REGION

REGION Network 17: **** 4.6 - Mashine Status - Indications **** Icon Animation 1
   // Icon Animation 1
   IF "TRUE" THEN
       "LSimpleIAnim"(I_SetPos := #I_Input1,
                      I_ResetPos := "FALSE",
                      I_Active := "FALSE",
                      I_Invisible := #I_Invisible1,
                      I_OutOfUse := "FALSE",
                      I_AlarmA := #Alarm1 AND #AlarmClass1_A,
                      I_AlarmB := #Alarm1 AND #AlarmClass1_B,
                      I_AlarmC := #Alarm1 AND #AlarmClass1_C,
                      I_AlarmD := #Alarm1 AND #AlarmClass1_D,
                      I_ManualMode := "FALSE",
                      I_FncSelInHMI := "FALSE",
                      H_IAnim => #H_IAnim1);
   END_IF;
END_REGION

REGION Network 18: **** 4.6 - Mashine Status - Indications **** Icon Animation 2
   // Icon Animation 2
   IF "TRUE" THEN
       "LSimpleIAnim"(I_SetPos := #I_Input2,
                      I_ResetPos := "FALSE",
                      I_Active := "FALSE",
                      I_Invisible := #I_Invisible2,
                      I_OutOfUse := "FALSE",
                      I_AlarmA := #Alarm2 AND #AlarmClass2_A,
                      I_AlarmB := #Alarm2 AND #AlarmClass2_B,
                      I_AlarmC := #Alarm2 AND #AlarmClass2_C,
                      I_AlarmD := #Alarm2 AND #AlarmClass2_D,
                      I_ManualMode := "FALSE",
                      I_FncSelInHMI := "FALSE",
                      H_IAnim => #H_IAnim2);
   END_IF;
END_REGION

REGION Network 19: **** 4.6 - Mashine Status - Indications **** Icon Animation 3
   // Icon Animation 3
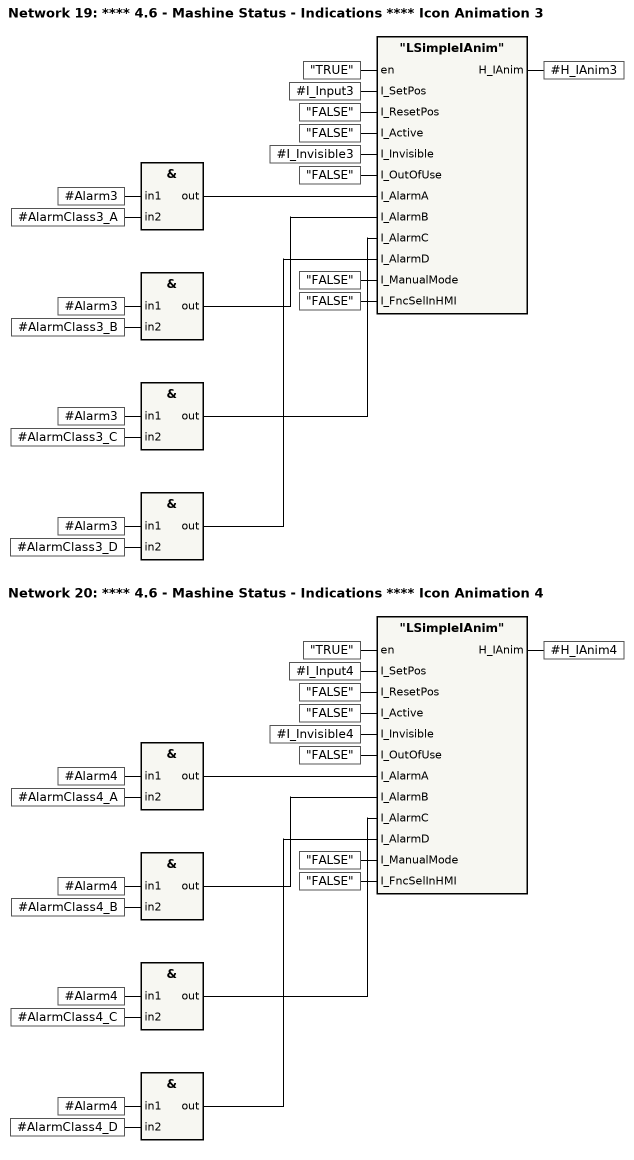
   IF "TRUE" THEN
       "LSimpleIAnim"(I_SetPos := #I_Input3,
                      I_ResetPos := "FALSE",
                      I_Active := "FALSE",
                      I_Invisible := #I_Invisible3,
                      I_OutOfUse := "FALSE",
                      I_AlarmA := #Alarm3 AND #AlarmClass3_A,
                      I_AlarmB := #Alarm3 AND #AlarmClass3_B,
                      I_AlarmC := #Alarm3 AND #AlarmClass3_C,
                      I_AlarmD := #Alarm3 AND #AlarmClass3_D,
                      I_ManualMode := "FALSE",
                      I_FncSelInHMI := "FALSE",
                      H_IAnim => #H_IAnim3);
   END_IF;
END_REGION

REGION Network 20: **** 4.6 - Mashine Status - Indications **** Icon Animation 4
   // Icon Animation 4
   IF "TRUE" THEN
       "LSimpleIAnim"(I_SetPos := #I_Input4,
                      I_ResetPos := "FALSE",
                      I_Active := "FALSE",
                      I_Invisible := #I_Invisible4,
                      I_OutOfUse := "FALSE",
                      I_AlarmA := #Alarm4 AND #AlarmClass4_A,
                      I_AlarmB := #Alarm4 AND #AlarmClass4_B,
                      I_AlarmC := #Alarm4 AND #AlarmClass4_C,
                      I_AlarmD := #Alarm4 AND #AlarmClass4_D,
                      I_ManualMode := "FALSE",
                      I_FncSelInHMI := "FALSE",
                      H_IAnim => #H_IAnim4);
   END_IF;
END_REGION

REGION Network 21: **** 4.6 - Mashine Status - Indications **** Icon Animation 5
   // Icon Animation 5
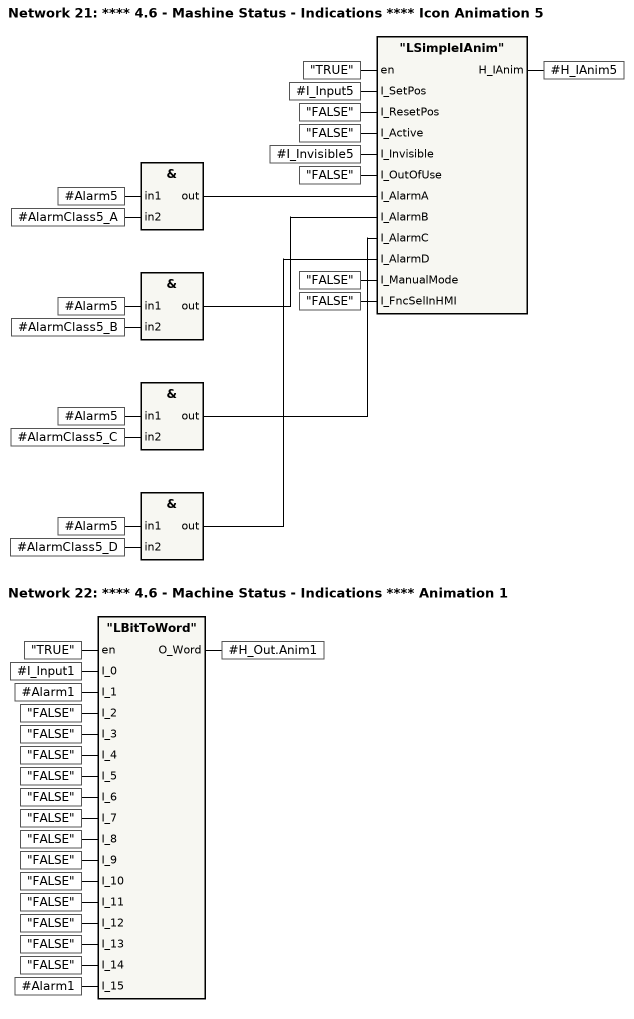
   IF "TRUE" THEN
       "LSimpleIAnim"(I_SetPos := #I_Input5,
                      I_ResetPos := "FALSE",
                      I_Active := "FALSE",
                      I_Invisible := #I_Invisible5,
                      I_OutOfUse := "FALSE",
                      I_AlarmA := #Alarm5 AND #AlarmClass5_A,
                      I_AlarmB := #Alarm5 AND #AlarmClass5_B,
                      I_AlarmC := #Alarm5 AND #AlarmClass5_C,
                      I_AlarmD := #Alarm5 AND #AlarmClass5_D,
                      I_ManualMode := "FALSE",
                      I_FncSelInHMI := "FALSE",
                      H_IAnim => #H_IAnim5);
   END_IF;
END_REGION

REGION Network 22: **** 4.6 - Machine Status - Indications **** Animation 1
   // Animation 1
   IF "TRUE" THEN
       "LBitToWord"(I_0 := #I_Input1,
                    I_1 := #Alarm1,
                    I_2 := "FALSE",
                    I_3 := "FALSE",
                    I_4 := "FALSE",
                    I_5 := "FALSE",
                    I_6 := "FALSE",
                    I_7 := "FALSE",
                    I_8 := "FALSE",
                    I_9 := "FALSE",
                    I_10 := "FALSE",
                    I_11 := "FALSE",
                    I_12 := "FALSE",
                    I_13 := "FALSE",
                    I_14 := "FALSE",
                    I_15 := #Alarm1,
                    O_Word => #H_Out.Anim1);
   END_IF;
END_REGION

REGION Network 23: **** 4.6 - Machine Status - Indications **** Animation 2
   // Animation 2
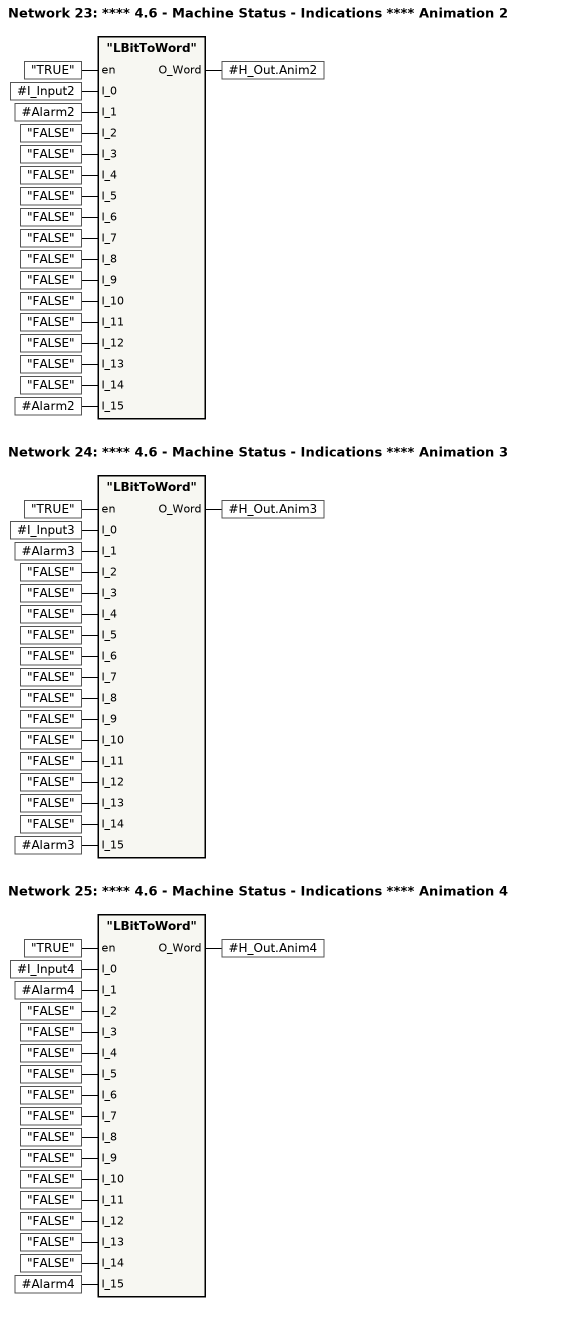
   IF "TRUE" THEN
       "LBitToWord"(I_0 := #I_Input2,
                    I_1 := #Alarm2,
                    I_2 := "FALSE",
                    I_3 := "FALSE",
                    I_4 := "FALSE",
                    I_5 := "FALSE",
                    I_6 := "FALSE",
                    I_7 := "FALSE",
                    I_8 := "FALSE",
                    I_9 := "FALSE",
                    I_10 := "FALSE",
                    I_11 := "FALSE",
                    I_12 := "FALSE",
                    I_13 := "FALSE",
                    I_14 := "FALSE",
                    I_15 := #Alarm2,
                    O_Word => #H_Out.Anim2);
   END_IF;
END_REGION

REGION Network 24: **** 4.6 - Machine Status - Indications **** Animation 3
   // Animation 3
   IF "TRUE" THEN
       "LBitToWord"(I_0 := #I_Input3,
                    I_1 := #Alarm3,
                    I_2 := "FALSE",
                    I_3 := "FALSE",
                    I_4 := "FALSE",
                    I_5 := "FALSE",
                    I_6 := "FALSE",
                    I_7 := "FALSE",
                    I_8 := "FALSE",
                    I_9 := "FALSE",
                    I_10 := "FALSE",
                    I_11 := "FALSE",
                    I_12 := "FALSE",
                    I_13 := "FALSE",
                    I_14 := "FALSE",
                    I_15 := #Alarm3,
                    O_Word => #H_Out.Anim3);
   END_IF;
END_REGION

REGION Network 25: **** 4.6 - Machine Status - Indications **** Animation 4
   // Animation 4
   IF "TRUE" THEN
       "LBitToWord"(I_0 := #I_Input4,
                    I_1 := #Alarm4,
                    I_2 := "FALSE",
                    I_3 := "FALSE",
                    I_4 := "FALSE",
                    I_5 := "FALSE",
                    I_6 := "FALSE",
                    I_7 := "FALSE",
                    I_8 := "FALSE",
                    I_9 := "FALSE",
                    I_10 := "FALSE",
                    I_11 := "FALSE",
                    I_12 := "FALSE",
                    I_13 := "FALSE",
                    I_14 := "FALSE",
                    I_15 := #Alarm4,
                    O_Word => #H_Out.Anim4);
   END_IF;
END_REGION

REGION Network 26: **** 4.6 - Machine Status - Indications **** Animation 5
   // Animation 5
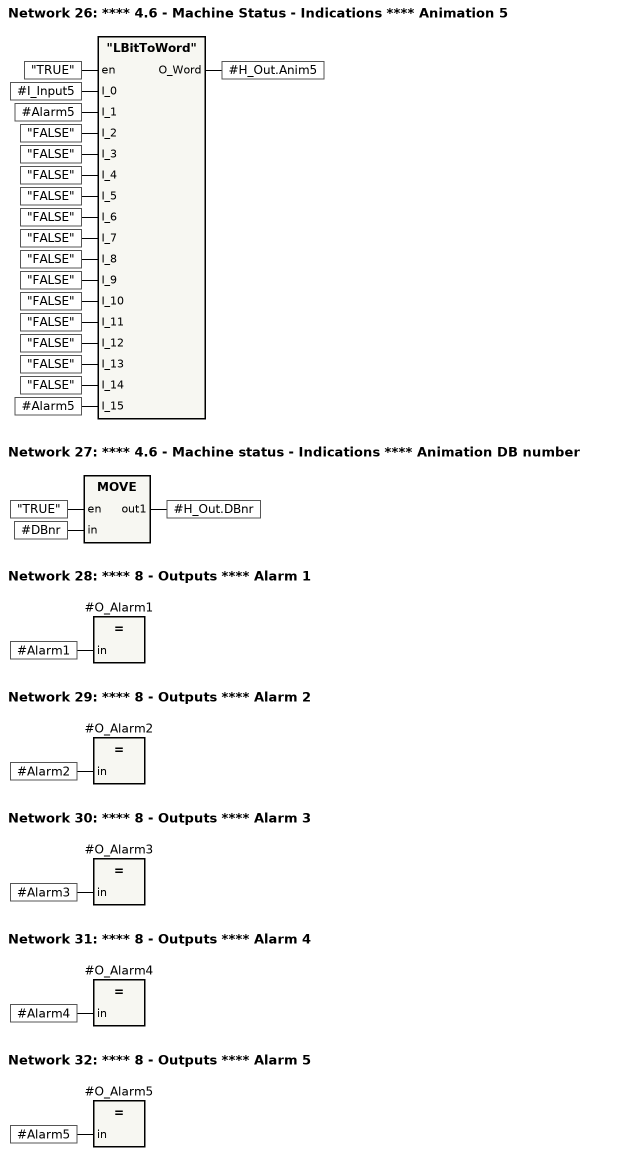
   IF "TRUE" THEN
       "LBitToWord"(I_0 := #I_Input5,
                    I_1 := #Alarm5,
                    I_2 := "FALSE",
                    I_3 := "FALSE",
                    I_4 := "FALSE",
                    I_5 := "FALSE",
                    I_6 := "FALSE",
                    I_7 := "FALSE",
                    I_8 := "FALSE",
                    I_9 := "FALSE",
                    I_10 := "FALSE",
                    I_11 := "FALSE",
                    I_12 := "FALSE",
                    I_13 := "FALSE",
                    I_14 := "FALSE",
                    I_15 := #Alarm5,
                    O_Word => #H_Out.Anim5);
   END_IF;
END_REGION

REGION Network 27: **** 4.6 - Machine status - Indications **** Animation DB number
   IF "TRUE" THEN #H_Out.DBnr := #DBnr; END_IF;
END_REGION

REGION Network 28: **** 8 - Outputs **** Alarm 1
   // Output of the Alarm 1
   #O_Alarm1 := #Alarm1;
END_REGION

REGION Network 29: **** 8 - Outputs **** Alarm 2
   // Output of the Alarm 2
   #O_Alarm2 := #Alarm2;
END_REGION

REGION Network 30: **** 8 - Outputs **** Alarm 3
   // Output of the Alarm 3
   #O_Alarm3 := #Alarm3;
END_REGION

REGION Network 31: **** 8 - Outputs **** Alarm 4
   // Output of the Alarm 4
   #O_Alarm4 := #Alarm4;
END_REGION

REGION Network 32: **** 8 - Outputs **** Alarm 5
   // Output of the Alarm 5
   #O_Alarm5 := #Alarm5;
END_REGION

REGION Network 33: **** 8 - Outputs **** Alarm AB Condition
   // Alarm AB condition
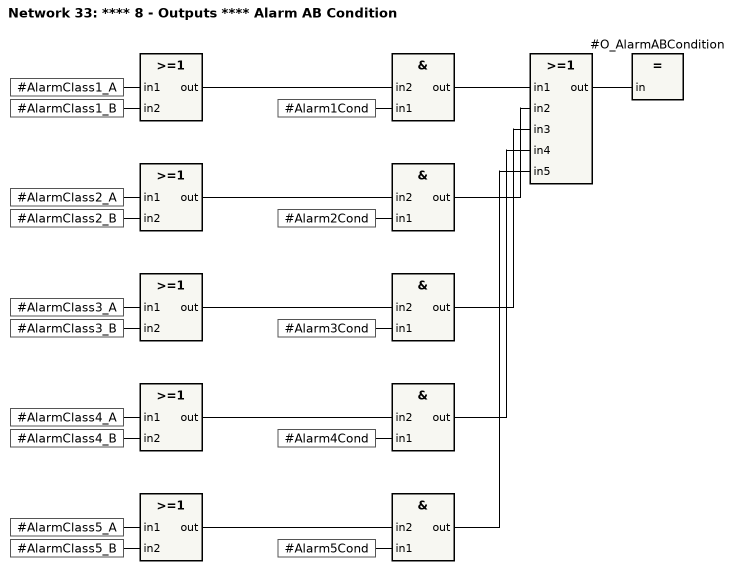
   #O_AlarmABCondition := ((#AlarmClass1_A OR #AlarmClass1_B) AND #Alarm1Cond) OR ((#AlarmClass2_A OR #AlarmClass2_B) AND #Alarm2Cond) OR ((#AlarmClass3_A OR #AlarmClass3_B) AND #Alarm3Cond) OR ((#AlarmClass4_A OR #AlarmClass4_B) AND #Alarm4Cond) OR ((#AlarmClass5_A OR #AlarmClass5_B) AND #Alarm5Cond);
END_REGION
END_FUNCTION_BLOCK

FUNCTION_BLOCK "LETAFuseCPC20PN"   // FB1406, FBD
TITLE = LETAFuseCPC20PN
{ S7_Optimized_Access := 'TRUE' }
AUTHOR : VCC
FAMILY : AlarmHnd
VERSION : 0.1
// stored: AutoNumber false, IsIECCheckEnabled false, IsRetainMemResEnabled false, MemoryReserve 100, SetENOAutomatically False, UDAEnableTagReadback false
   VAR_INPUT
      I_NewShift { ExternalAccessible := 'False'; ExternalVisible := 'False'; ExternalWritable := 'False'} : Bool;   // NewShift / Morning shift
      I_EnableAlarm { ExternalAccessible := 'False'; ExternalVisible := 'False'; ExternalWritable := 'False'} : Bool := TRUE;   // Enable Alarm from upper level
      C_HWInput { ExternalAccessible := 'False'; ExternalVisible := 'False'; ExternalWritable := 'False'} : HW_IO;   // Slot ID from CPC20PN
      C_Block1_TotalCurrent { ExternalAccessible := 'False'; ExternalVisible := 'False'; ExternalWritable := 'False'} : HW_IO;   // Base Module Slot ID Total Current, 0=not in use.
      C_Block1_StatusControl { ExternalAccessible := 'False'; ExternalVisible := 'False'; ExternalWritable := 'False'} : HW_IO;   // Base Module Slot ID Status / Control, 0=not in use.
      "C_Block1_MeasurementU/I" { ExternalAccessible := 'False'; ExternalVisible := 'False'; ExternalWritable := 'False'} : HW_IO;   // Base Module Slot ID Measurement UI, 0=not in use.
      C_Block2_TotalCurrent { ExternalAccessible := 'False'; ExternalVisible := 'False'; ExternalWritable := 'False'} : HW_IO;   // Extension Module Slot ID Total Current, 0=not in use.
      C_Block2_StatusControl { ExternalAccessible := 'False'; ExternalVisible := 'False'; ExternalWritable := 'False'} : HW_IO;   // Extension Module Slot ID Status / Control, 0=not in use.
      "C_Block2_MeasurementU/I" { ExternalAccessible := 'False'; ExternalVisible := 'False'; ExternalWritable := 'False'} : HW_IO;   // Extension Module Slot ID Measurement UI, 0=not in use.
      C_Config { ExternalAccessible := 'False'; ExternalVisible := 'False'; ExternalWritable := 'False'} : "ETAFuseCPC20PNConfig";   // Config
   END_VAR
   VAR_OUTPUT
      O_AlarmABCondition { ExternalAccessible := 'False'; ExternalVisible := 'False'; ExternalWritable := 'False'} : Bool;   // Alarm AB Condition
      O_AlarmA { ExternalAccessible := 'False'; ExternalVisible := 'False'; ExternalWritable := 'False'} : Bool;   // Alarm A
      O_AlarmB { ExternalAccessible := 'False'; ExternalVisible := 'False'; ExternalWritable := 'False'} : Bool;   // Alarm B
      O_AlarmC { ExternalAccessible := 'False'; ExternalVisible := 'False'; ExternalWritable := 'False'} : Bool;   // Alarm C
      O_AlarmD { ExternalAccessible := 'False'; ExternalVisible := 'False'; ExternalWritable := 'False'} : Bool;   // Alarm D
      H_AlarmDWord { ExternalAccessible := 'False'; ExternalVisible := 'False'; ExternalWritable := 'False'} : DWord;   // HMI Animation
   END_VAR
   VAR_IN_OUT
      IO_ETAFuseData : "ETAFuseData";   // ETA fuse status
      H_HMI : "H_HMI";   // Animation
      H_ETAFuseCPC20PN : "H_ETAFuseCPC20PN";   // Animation
   END_VAR
   VAR
      AC_StatusCPC20_Bit0 { ExternalAccessible := 'False'; ExternalVisible := 'False'; ExternalWritable := 'False'} : Bool;   // No configuration data available
      AC_StatusCPC20_Bit1 { ExternalAccessible := 'False'; ExternalVisible := 'False'; ExternalWritable := 'False'} : Bool;   // Invalid configuration data
      AC_StatusCPC20_Bit4 { ExternalAccessible := 'False'; ExternalVisible := 'False'; ExternalWritable := 'False'} : Bool;   // Command buffer overflow
      AC_StatusCPC20_Bit7 { ExternalAccessible := 'False'; ExternalVisible := 'False'; ExternalWritable := 'False'} : Bool;   // No communication with at least one PWR board
      AC_StatusCPC20_Bit9 { ExternalAccessible := 'False'; ExternalVisible := 'False'; ExternalWritable := 'False'} : Bool;   // CPC tempory error
      AC_StatusCPC20_Bit10 { ExternalAccessible := 'False'; ExternalVisible := 'False'; ExternalWritable := 'False'} : Bool;   // CPC hardware error
      AC_ReadNomCurr { ExternalAccessible := 'False'; ExternalVisible := 'False'; ExternalWritable := 'False'} : Bool;   // Overtime Reading of nominal current
      AlarmABCondition { ExternalAccessible := 'False'; ExternalVisible := 'False'; ExternalWritable := 'False'} : Bool;   // Alarm AB Condition
      AlarmA { ExternalAccessible := 'False'; ExternalVisible := 'False'; ExternalWritable := 'False'} : Bool;   // Alarm A
      AlarmB { ExternalAccessible := 'False'; ExternalVisible := 'False'; ExternalWritable := 'False'} : Bool;   // Alarm B
      AlarmC { ExternalAccessible := 'False'; ExternalVisible := 'False'; ExternalWritable := 'False'} : Bool;   // Alarm C
      AlarmD { ExternalAccessible := 'False'; ExternalVisible := 'False'; ExternalWritable := 'False'} : Bool;   // Alarm D
      ReadNominalCurrentActive { ExternalAccessible := 'False'; ExternalVisible := 'False'; ExternalWritable := 'False'} : Bool;   // Reading of nominal current is active
      EnableAlarm { ExternalAccessible := 'False'; ExternalVisible := 'False'; ExternalWritable := 'False'} : Bool;   // Enable Alarm from upper level
   END_VAR
   VAR RETAIN
      H_ReadNomCurr { ExternalAccessible := 'False'; ExternalVisible := 'False'; ExternalWritable := 'False'} : Bool;   // HMI Command - Read nominal current
      H_CancelReadNomCurr { ExternalAccessible := 'False'; ExternalVisible := 'False'; ExternalWritable := 'False'} : Bool;   // HMI Command - Cancel Read nominal current
   END_VAR
   VAR
      H_UpChannel { ExternalAccessible := 'False'; ExternalVisible := 'False'; ExternalWritable := 'False'} : Bool;   // HMI Command - UP channel selection
      H_DownChannel { ExternalAccessible := 'False'; ExternalVisible := 'False'; ExternalWritable := 'False'} : Bool;   // HMI Command - DOWN channel selection
      H_SwitchON { ExternalAccessible := 'False'; ExternalVisible := 'False'; ExternalWritable := 'False'} : Bool;   // HMICmd / HMI Command - Switch On
      H_SwitchOFF { ExternalAccessible := 'False'; ExternalVisible := 'False'; ExternalWritable := 'False'} : Bool;   // HMICmd / HMI Command - Switch Off
      H_Transfer { ExternalAccessible := 'False'; ExternalVisible := 'False'; ExternalWritable := 'False'} : Bool;   // HMICmd / HMI Command - Transfer
      H_Reset { ExternalAccessible := 'False'; ExternalVisible := 'False'; ExternalWritable := 'False'} : Bool;   // HMICmd / HMI Command - Reset
      _ETAFuseCPC20PNSub { ExternalAccessible := 'False'; ExternalVisible := 'False'; ExternalWritable := 'False'} : "LETAFuseCPC20PNSub";   // FB
   END_VAR
   VAR DB_SPECIFIC
      T_ResetControl { ExternalAccessible := 'False'; ExternalVisible := 'False'; ExternalWritable := 'False'} : TON_TIME;   // Timer
      T_EnableAlarm { ExternalAccessible := 'False'; ExternalVisible := 'False'; ExternalWritable := 'False'} : TON_TIME;   // Timer
   END_VAR
   VAR
      Edge { ExternalAccessible := 'False'; ExternalVisible := 'False'; ExternalWritable := 'False'} : Array[0..10] of Bool;   // Edge
   END_VAR
   VAR_TEMP   // added for the SCL form of the ladder/FBD networks
      _w1 : Bool;
      _w2 : Bool;
   END_VAR
BEGIN

REGION Network 1: **** 1 - Inputs **** Extract The Commands From HMI
   // Extract The Commands From HMI
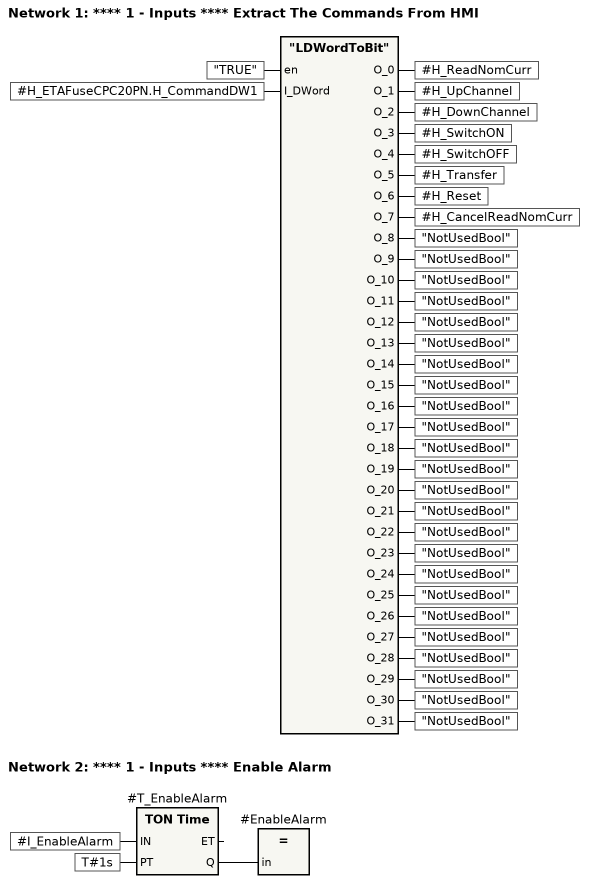
   IF "TRUE" THEN
       "LDWordToBit"(I_DWord := #H_ETAFuseCPC20PN.H_CommandDW1,
                     O_0 => #H_ReadNomCurr,
                     O_1 => #H_UpChannel,
                     O_2 => #H_DownChannel,
                     O_3 => #H_SwitchON,
                     O_4 => #H_SwitchOFF,
                     O_5 => #H_Transfer,
                     O_6 => #H_Reset,
                     O_7 => #H_CancelReadNomCurr,
                     O_8 => "NotUsedBool",
                     O_9 => "NotUsedBool",
                     O_10 => "NotUsedBool",
                     O_11 => "NotUsedBool",
                     O_12 => "NotUsedBool",
                     O_13 => "NotUsedBool",
                     O_14 => "NotUsedBool",
                     O_15 => "NotUsedBool",
                     O_16 => "NotUsedBool",
                     O_17 => "NotUsedBool",
                     O_18 => "NotUsedBool",
                     O_19 => "NotUsedBool",
                     O_20 => "NotUsedBool",
                     O_21 => "NotUsedBool",
                     O_22 => "NotUsedBool",
                     O_23 => "NotUsedBool",
                     O_24 => "NotUsedBool",
                     O_25 => "NotUsedBool",
                     O_26 => "NotUsedBool",
                     O_27 => "NotUsedBool",
                     O_28 => "NotUsedBool",
                     O_29 => "NotUsedBool",
                     O_30 => "NotUsedBool",
                     O_31 => "NotUsedBool");
   END_IF;
END_REGION

REGION Network 2: **** 1 - Inputs **** Enable Alarm
   #T_EnableAlarm(IN := #I_EnableAlarm, PT := T#1s);   // TON
   #EnableAlarm := #T_EnableAlarm.Q;
END_REGION

REGION Network 3: **** 4.3 - Machine status - Operator Selection **** Selected Channel
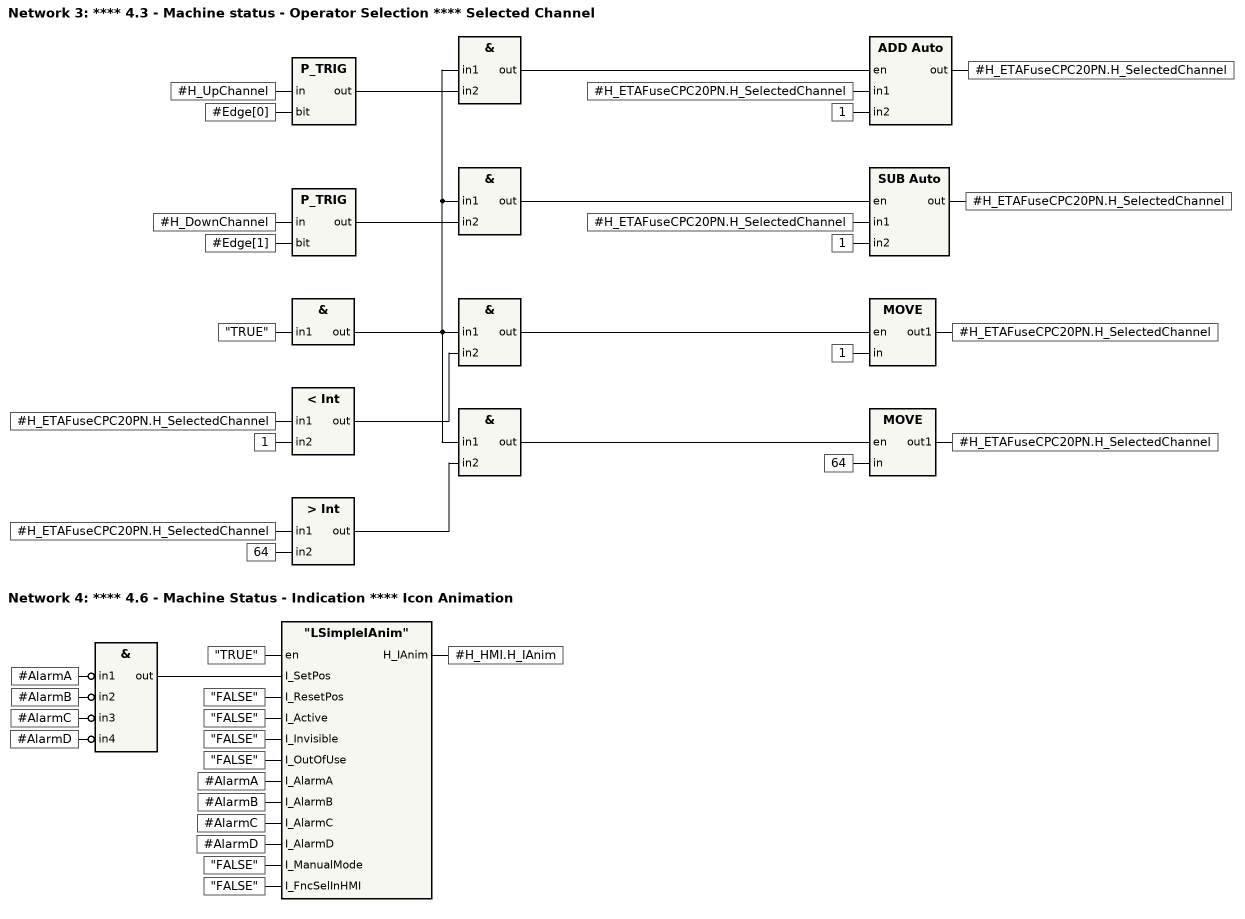
   #_w1 := #H_UpChannel AND NOT #Edge[0];   // rising edge
   #Edge[0] := #H_UpChannel;
   IF "TRUE" AND #_w1 THEN
       #H_ETAFuseCPC20PN.H_SelectedChannel := #H_ETAFuseCPC20PN.H_SelectedChannel + 1;
   END_IF;
   #_w2 := #H_DownChannel AND NOT #Edge[1];   // rising edge
   #Edge[1] := #H_DownChannel;
   IF "TRUE" AND #_w2 THEN
       #H_ETAFuseCPC20PN.H_SelectedChannel := #H_ETAFuseCPC20PN.H_SelectedChannel - 1;
   END_IF;
   IF "TRUE" AND (#H_ETAFuseCPC20PN.H_SelectedChannel < 1) THEN
       #H_ETAFuseCPC20PN.H_SelectedChannel := 1;
   END_IF;
   IF "TRUE" AND (#H_ETAFuseCPC20PN.H_SelectedChannel > 64) THEN
       #H_ETAFuseCPC20PN.H_SelectedChannel := 64;
   END_IF;
END_REGION

REGION Network 4: **** 4.6 - Machine Status - Indication **** Icon Animation
   // Icon Animation
   IF "TRUE" THEN
       "LSimpleIAnim"(I_SetPos := NOT #AlarmA AND NOT #AlarmB AND NOT #AlarmC AND NOT #AlarmD,
                      I_ResetPos := "FALSE",
                      I_Active := "FALSE",
                      I_Invisible := "FALSE",
                      I_OutOfUse := "FALSE",
                      I_AlarmA := #AlarmA,
                      I_AlarmB := #AlarmB,
                      I_AlarmC := #AlarmC,
                      I_AlarmD := #AlarmD,
                      I_ManualMode := "FALSE",
                      I_FncSelInHMI := "FALSE",
                      H_IAnim => #H_HMI.H_IAnim);
   END_IF;
END_REGION

REGION Network 5: **** 4.6 - Machine Status - Indication **** Animation
   // Animation
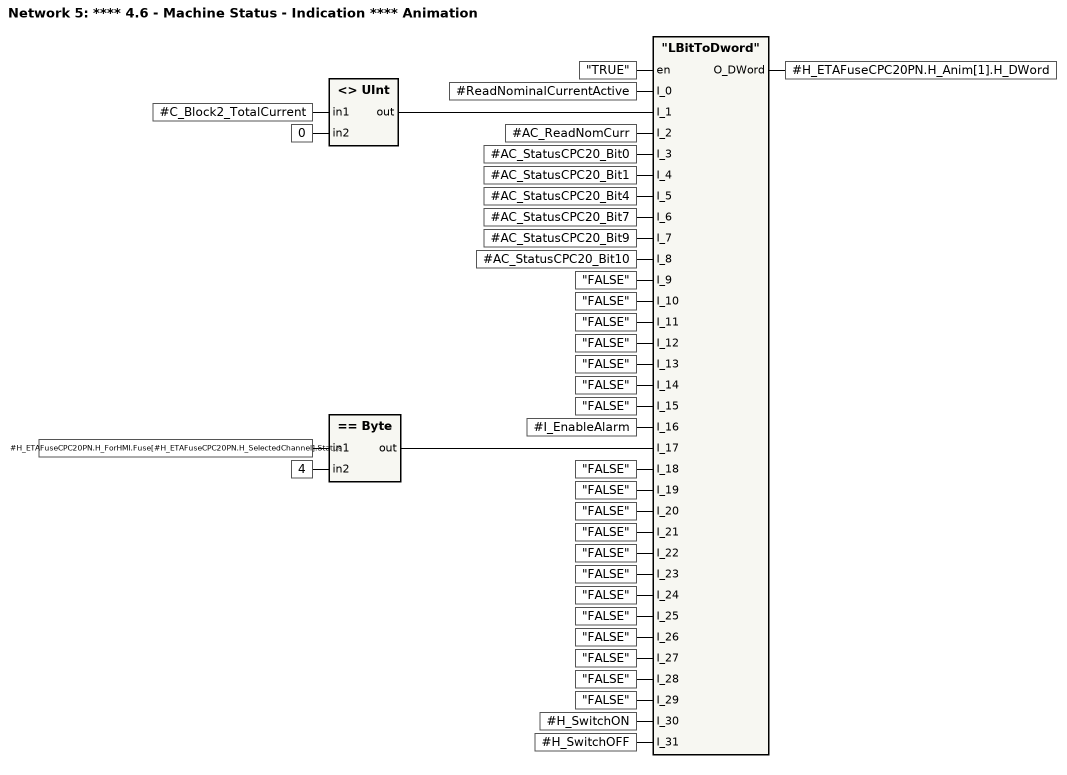
   IF "TRUE" THEN
       "LBitToDword"(I_0 := #ReadNominalCurrentActive,
                     I_1 := #C_Block2_TotalCurrent <> 0,
                     I_2 := #AC_ReadNomCurr,
                     I_3 := #AC_StatusCPC20_Bit0,
                     I_4 := #AC_StatusCPC20_Bit1,
                     I_5 := #AC_StatusCPC20_Bit4,
                     I_6 := #AC_StatusCPC20_Bit7,
                     I_7 := #AC_StatusCPC20_Bit9,
                     I_8 := #AC_StatusCPC20_Bit10,
                     I_9 := "FALSE",
                     I_10 := "FALSE",
                     I_11 := "FALSE",
                     I_12 := "FALSE",
                     I_13 := "FALSE",
                     I_14 := "FALSE",
                     I_15 := "FALSE",
                     I_16 := #I_EnableAlarm,
                     I_17 := #H_ETAFuseCPC20PN.H_ForHMI.Fuse[#H_ETAFuseCPC20PN.H_SelectedChannel].Status = 4,
                     I_18 := "FALSE",
                     I_19 := "FALSE",
                     I_20 := "FALSE",
                     I_21 := "FALSE",
                     I_22 := "FALSE",
                     I_23 := "FALSE",
                     I_24 := "FALSE",
                     I_25 := "FALSE",
                     I_26 := "FALSE",
                     I_27 := "FALSE",
                     I_28 := "FALSE",
                     I_29 := "FALSE",
                     I_30 := #H_SwitchON,
                     I_31 := #H_SwitchOFF,
                     O_DWord => #H_ETAFuseCPC20PN.H_Anim[1].H_DWord);
   END_IF;
END_REGION

REGION Network 6: **** 4.6 - Machine Status - Indication **** Animation
   // Animation
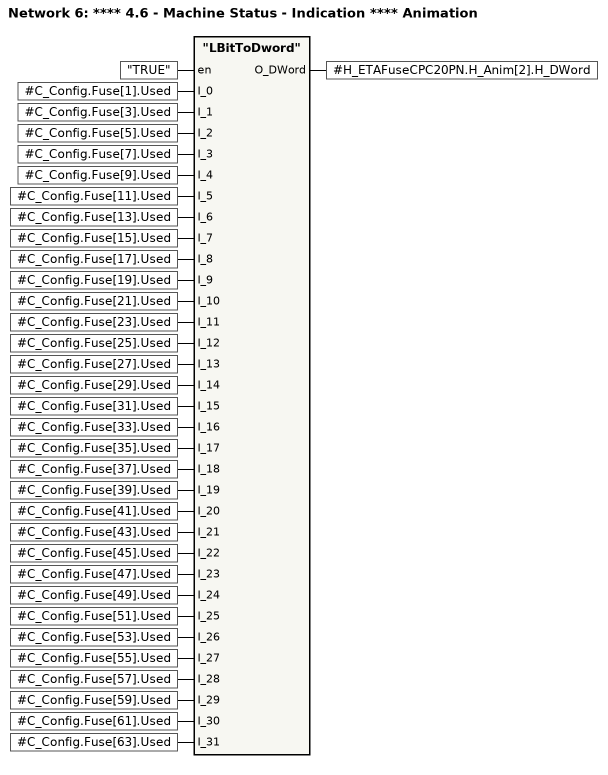
   IF "TRUE" THEN
       "LBitToDword"(I_0 := #C_Config.Fuse[1].Used,
                     I_1 := #C_Config.Fuse[3].Used,
                     I_2 := #C_Config.Fuse[5].Used,
                     I_3 := #C_Config.Fuse[7].Used,
                     I_4 := #C_Config.Fuse[9].Used,
                     I_5 := #C_Config.Fuse[11].Used,
                     I_6 := #C_Config.Fuse[13].Used,
                     I_7 := #C_Config.Fuse[15].Used,
                     I_8 := #C_Config.Fuse[17].Used,
                     I_9 := #C_Config.Fuse[19].Used,
                     I_10 := #C_Config.Fuse[21].Used,
                     I_11 := #C_Config.Fuse[23].Used,
                     I_12 := #C_Config.Fuse[25].Used,
                     I_13 := #C_Config.Fuse[27].Used,
                     I_14 := #C_Config.Fuse[29].Used,
                     I_15 := #C_Config.Fuse[31].Used,
                     I_16 := #C_Config.Fuse[33].Used,
                     I_17 := #C_Config.Fuse[35].Used,
                     I_18 := #C_Config.Fuse[37].Used,
                     I_19 := #C_Config.Fuse[39].Used,
                     I_20 := #C_Config.Fuse[41].Used,
                     I_21 := #C_Config.Fuse[43].Used,
                     I_22 := #C_Config.Fuse[45].Used,
                     I_23 := #C_Config.Fuse[47].Used,
                     I_24 := #C_Config.Fuse[49].Used,
                     I_25 := #C_Config.Fuse[51].Used,
                     I_26 := #C_Config.Fuse[53].Used,
                     I_27 := #C_Config.Fuse[55].Used,
                     I_28 := #C_Config.Fuse[57].Used,
                     I_29 := #C_Config.Fuse[59].Used,
                     I_30 := #C_Config.Fuse[61].Used,
                     I_31 := #C_Config.Fuse[63].Used,
                     O_DWord => #H_ETAFuseCPC20PN.H_Anim[2].H_DWord);
   END_IF;
END_REGION

REGION Network 7: **** 4.6 - Machine Status - Indication **** Animation
   // Animation
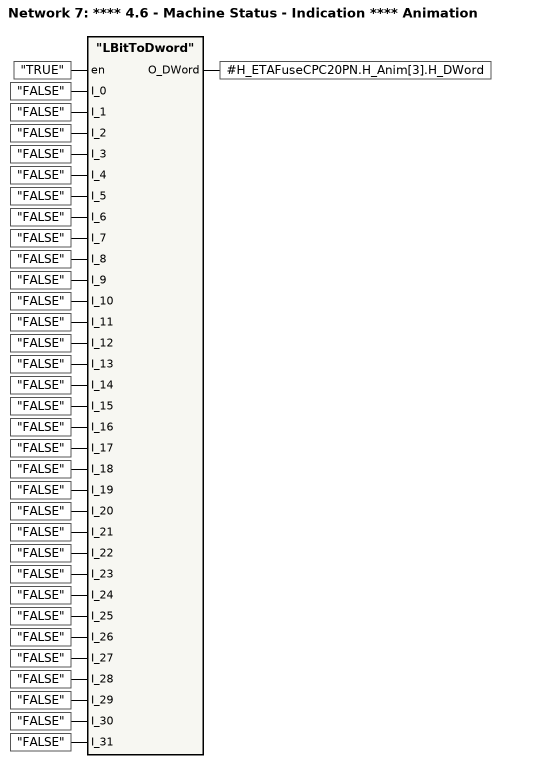
   IF "TRUE" THEN
       "LBitToDword"(I_0 := "FALSE",
                     I_1 := "FALSE",
                     I_2 := "FALSE",
                     I_3 := "FALSE",
                     I_4 := "FALSE",
                     I_5 := "FALSE",
                     I_6 := "FALSE",
                     I_7 := "FALSE",
                     I_8 := "FALSE",
                     I_9 := "FALSE",
                     I_10 := "FALSE",
                     I_11 := "FALSE",
                     I_12 := "FALSE",
                     I_13 := "FALSE",
                     I_14 := "FALSE",
                     I_15 := "FALSE",
                     I_16 := "FALSE",
                     I_17 := "FALSE",
                     I_18 := "FALSE",
                     I_19 := "FALSE",
                     I_20 := "FALSE",
                     I_21 := "FALSE",
                     I_22 := "FALSE",
                     I_23 := "FALSE",
                     I_24 := "FALSE",
                     I_25 := "FALSE",
                     I_26 := "FALSE",
                     I_27 := "FALSE",
                     I_28 := "FALSE",
                     I_29 := "FALSE",
                     I_30 := "FALSE",
                     I_31 := "FALSE",
                     O_DWord => #H_ETAFuseCPC20PN.H_Anim[3].H_DWord);
   END_IF;
END_REGION

REGION Network 8: **** 4.6 - Machine Status - Indication **** Animation
   // Animation
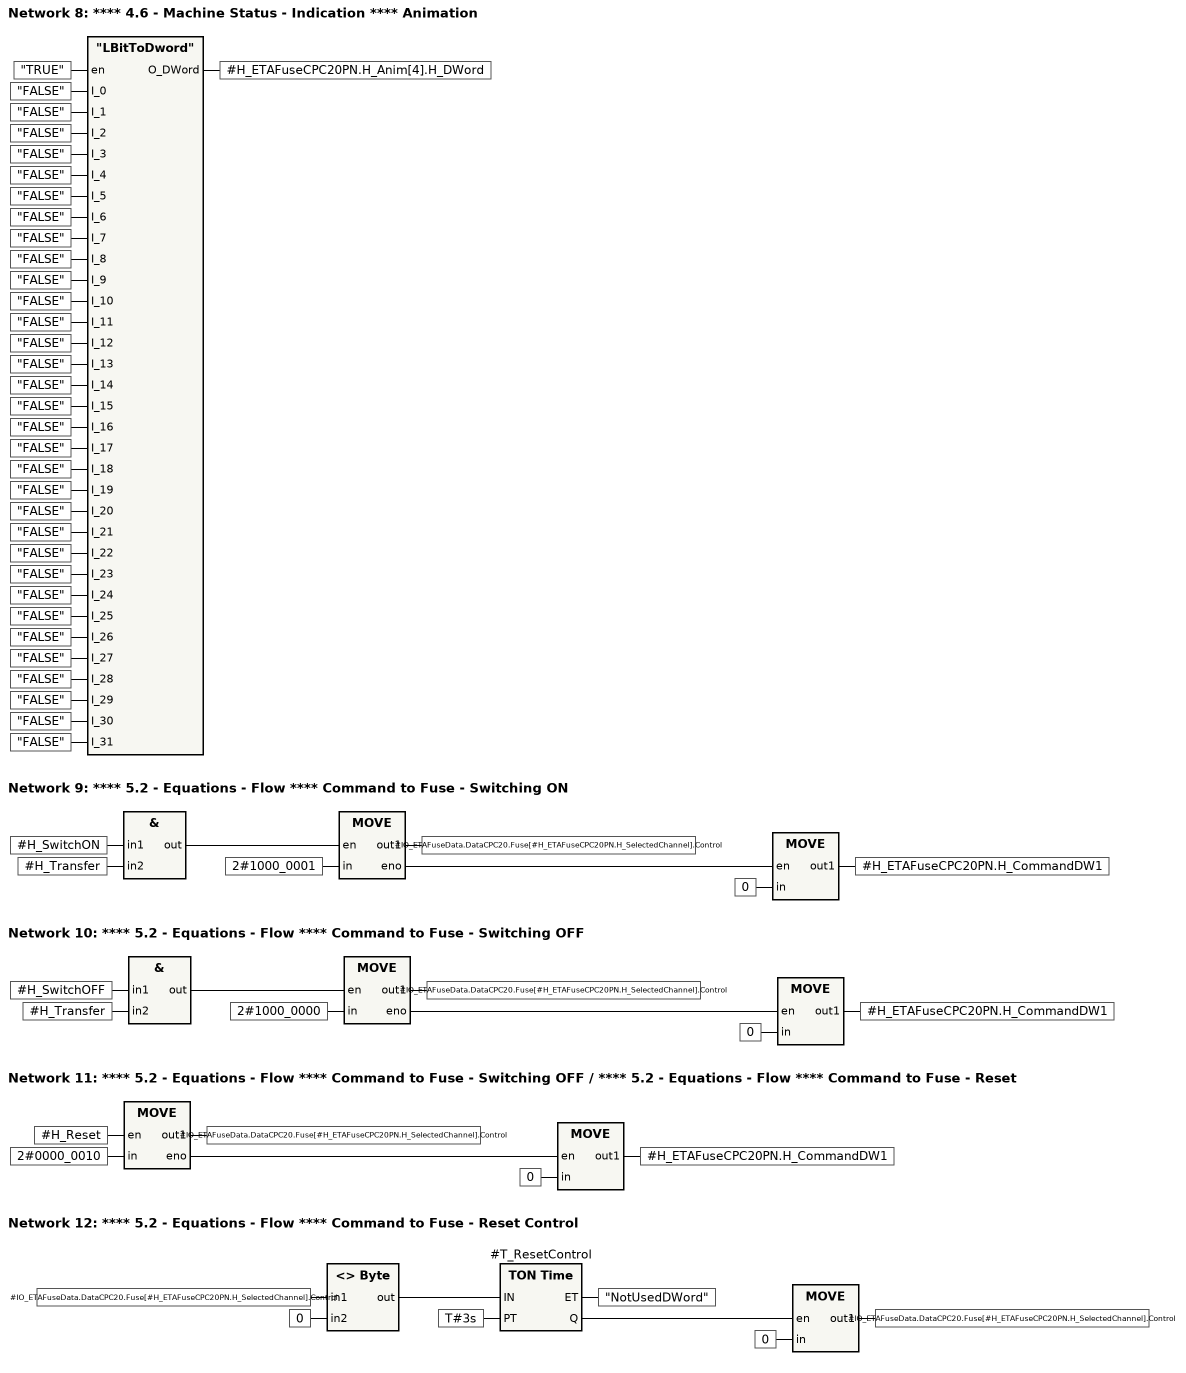
   IF "TRUE" THEN
       "LBitToDword"(I_0 := "FALSE",
                     I_1 := "FALSE",
                     I_2 := "FALSE",
                     I_3 := "FALSE",
                     I_4 := "FALSE",
                     I_5 := "FALSE",
                     I_6 := "FALSE",
                     I_7 := "FALSE",
                     I_8 := "FALSE",
                     I_9 := "FALSE",
                     I_10 := "FALSE",
                     I_11 := "FALSE",
                     I_12 := "FALSE",
                     I_13 := "FALSE",
                     I_14 := "FALSE",
                     I_15 := "FALSE",
                     I_16 := "FALSE",
                     I_17 := "FALSE",
                     I_18 := "FALSE",
                     I_19 := "FALSE",
                     I_20 := "FALSE",
                     I_21 := "FALSE",
                     I_22 := "FALSE",
                     I_23 := "FALSE",
                     I_24 := "FALSE",
                     I_25 := "FALSE",
                     I_26 := "FALSE",
                     I_27 := "FALSE",
                     I_28 := "FALSE",
                     I_29 := "FALSE",
                     I_30 := "FALSE",
                     I_31 := "FALSE",
                     O_DWord => #H_ETAFuseCPC20PN.H_Anim[4].H_DWord);
   END_IF;
END_REGION

REGION Network 9: **** 5.2 - Equations - Flow **** Command to Fuse - Switching ON
   // Switching ON
   // ENO of a box is taken as its EN; it also drops when the box reports an error
   IF #H_SwitchON AND #H_Transfer THEN
       #IO_ETAFuseData.DataCPC20.Fuse[#H_ETAFuseCPC20PN.H_SelectedChannel].Control := 2#1000_0001;
       #H_ETAFuseCPC20PN.H_CommandDW1 := 0;
   END_IF;
END_REGION

REGION Network 10: **** 5.2 - Equations - Flow **** Command to Fuse - Switching OFF
   // Switching OFF
   // ENO of a box is taken as its EN; it also drops when the box reports an error
   IF #H_SwitchOFF AND #H_Transfer THEN
       #IO_ETAFuseData.DataCPC20.Fuse[#H_ETAFuseCPC20PN.H_SelectedChannel].Control := 2#1000_0000;
       #H_ETAFuseCPC20PN.H_CommandDW1 := 0;
   END_IF;
END_REGION

REGION Network 11: **** 5.2 - Equations - Flow **** Command to Fuse - Switching OFF / **** 5.2 - Equations - Flow **** Command to Fuse - Reset
   // Switching OFF / Reset
   // ENO of a box is taken as its EN; it also drops when the box reports an error
   IF #H_Reset THEN
       #IO_ETAFuseData.DataCPC20.Fuse[#H_ETAFuseCPC20PN.H_SelectedChannel].Control := 2#0000_0010;
       #H_ETAFuseCPC20PN.H_CommandDW1 := 0;
   END_IF;
END_REGION

REGION Network 12: **** 5.2 - Equations - Flow **** Command to Fuse - Reset Control
   #T_ResetControl(IN := #IO_ETAFuseData.DataCPC20.Fuse[#H_ETAFuseCPC20PN.H_SelectedChannel].Control <> 0,   // TON
                   PT := T#3s,
                   ET => "NotUsedDWord");
   IF #T_ResetControl.Q THEN
       #IO_ETAFuseData.DataCPC20.Fuse[#H_ETAFuseCPC20PN.H_SelectedChannel].Control := 0;
   END_IF;
END_REGION

REGION Network 13: **** 7.1 - Submodule - Non-Machine **** ETA CPC20 PN
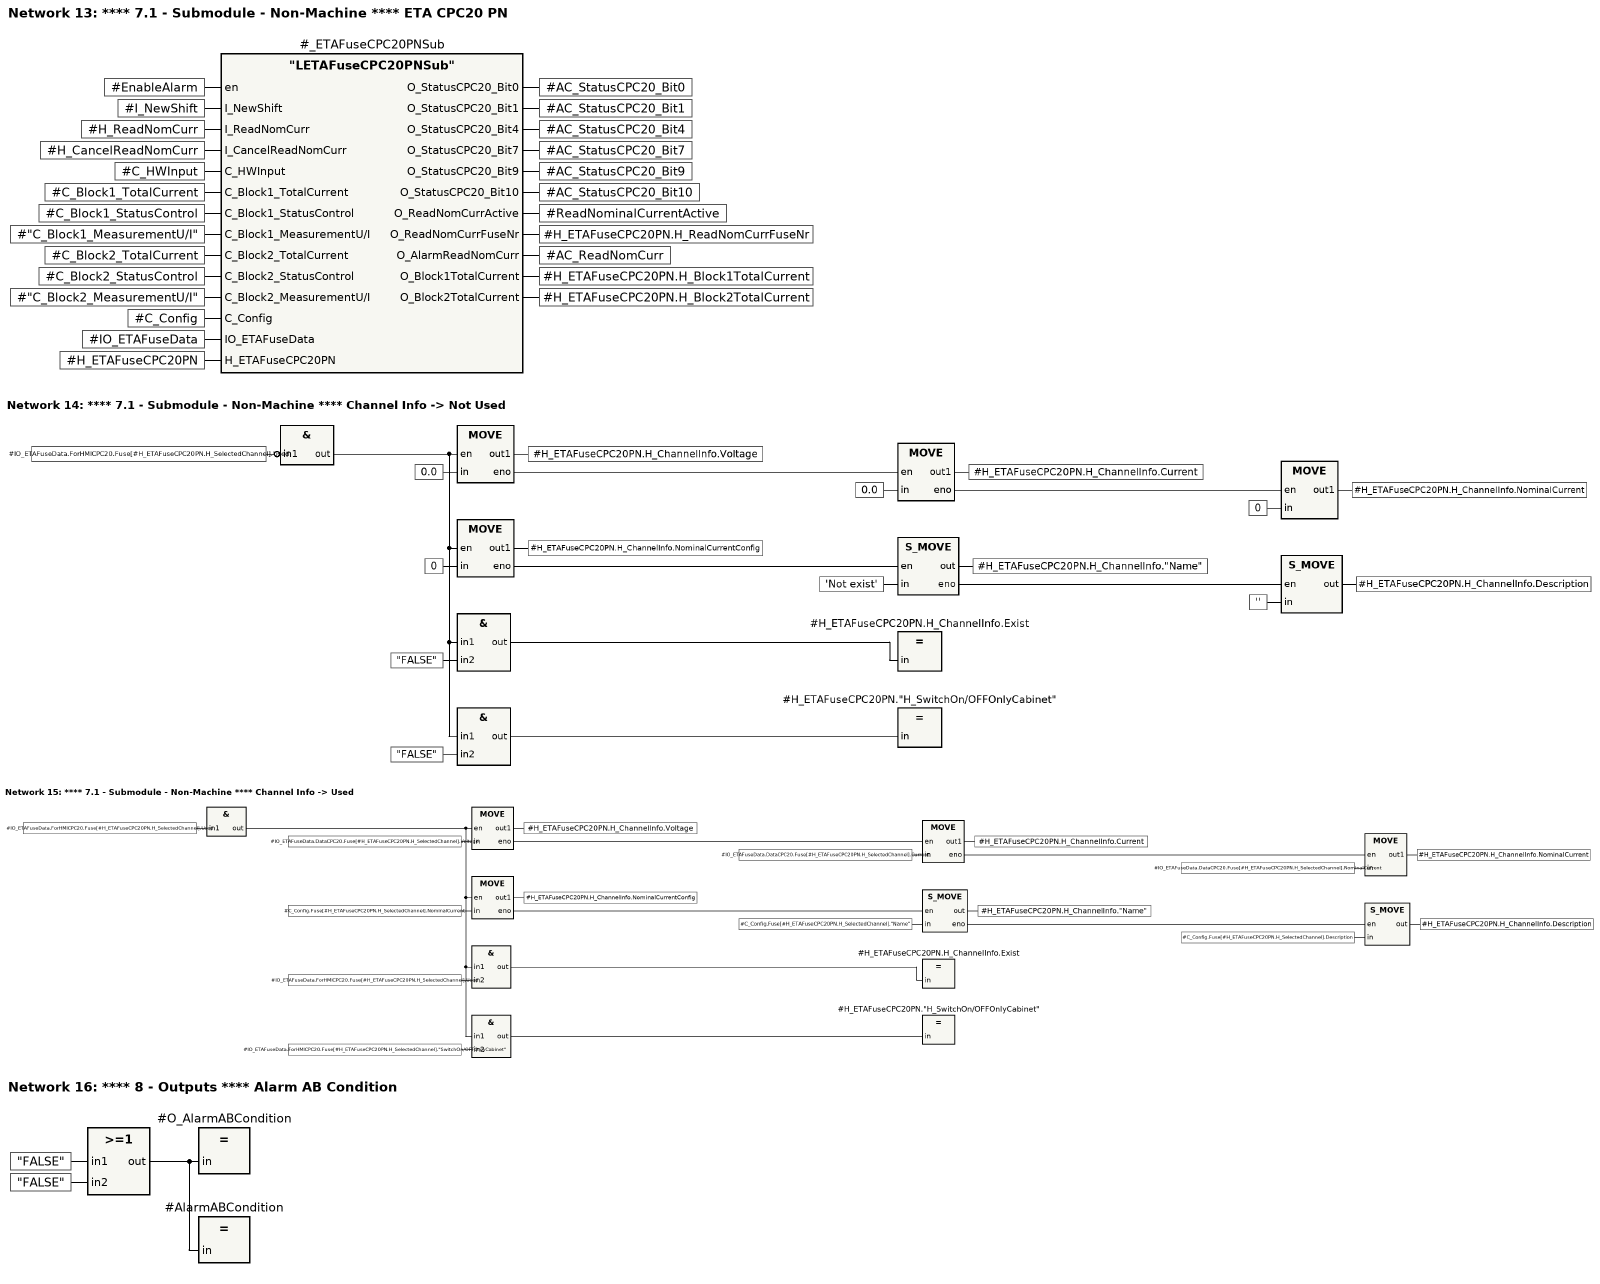
   IF #EnableAlarm THEN
       #_ETAFuseCPC20PNSub(I_NewShift := #I_NewShift,   // "LETAFuseCPC20PNSub"
                           I_ReadNomCurr := #H_ReadNomCurr,
                           I_CancelReadNomCurr := #H_CancelReadNomCurr,
                           C_HWInput := #C_HWInput,
                           C_Block1_TotalCurrent := #C_Block1_TotalCurrent,
                           C_Block1_StatusControl := #C_Block1_StatusControl,
                           "C_Block1_MeasurementU/I" := #"C_Block1_MeasurementU/I",
                           C_Block2_TotalCurrent := #C_Block2_TotalCurrent,
                           C_Block2_StatusControl := #C_Block2_StatusControl,
                           "C_Block2_MeasurementU/I" := #"C_Block2_MeasurementU/I",
                           C_Config := #C_Config,
                           IO_ETAFuseData := #IO_ETAFuseData,
                           H_ETAFuseCPC20PN := #H_ETAFuseCPC20PN,
                           O_StatusCPC20_Bit0 => #AC_StatusCPC20_Bit0,
                           O_StatusCPC20_Bit1 => #AC_StatusCPC20_Bit1,
                           O_StatusCPC20_Bit4 => #AC_StatusCPC20_Bit4,
                           O_StatusCPC20_Bit7 => #AC_StatusCPC20_Bit7,
                           O_StatusCPC20_Bit9 => #AC_StatusCPC20_Bit9,
                           O_StatusCPC20_Bit10 => #AC_StatusCPC20_Bit10,
                           O_ReadNomCurrActive => #ReadNominalCurrentActive,
                           O_ReadNomCurrFuseNr => #H_ETAFuseCPC20PN.H_ReadNomCurrFuseNr,
                           O_AlarmReadNomCurr => #AC_ReadNomCurr,
                           O_Block1TotalCurrent => #H_ETAFuseCPC20PN.H_Block1TotalCurrent,
                           O_Block2TotalCurrent => #H_ETAFuseCPC20PN.H_Block2TotalCurrent);
   END_IF;
END_REGION

REGION Network 14: **** 7.1 - Submodule - Non-Machine **** Channel Info -> Not Used
   #_w1 := NOT #IO_ETAFuseData.ForHMICPC20.Fuse[#H_ETAFuseCPC20PN.H_SelectedChannel].Used;
   IF #_w1 THEN
       #H_ETAFuseCPC20PN.H_ChannelInfo.Voltage := 0.0;
       #H_ETAFuseCPC20PN.H_ChannelInfo.Current := 0.0;
       #H_ETAFuseCPC20PN.H_ChannelInfo.NominalCurrent := 0;
       #H_ETAFuseCPC20PN.H_ChannelInfo.NominalCurrentConfig := 0;
       #H_ETAFuseCPC20PN.H_ChannelInfo."Name" := 'Not exist';
       #H_ETAFuseCPC20PN.H_ChannelInfo.Description := '';
   END_IF;
   #H_ETAFuseCPC20PN.H_ChannelInfo.Exist := #_w1 AND "FALSE";
   #H_ETAFuseCPC20PN."H_SwitchOn/OFFOnlyCabinet" := #_w1 AND "FALSE";
END_REGION

REGION Network 15: **** 7.1 - Submodule - Non-Machine **** Channel Info -> Used
   IF #IO_ETAFuseData.ForHMICPC20.Fuse[#H_ETAFuseCPC20PN.H_SelectedChannel].Used THEN
       #H_ETAFuseCPC20PN.H_ChannelInfo.Voltage := #IO_ETAFuseData.DataCPC20.Fuse[#H_ETAFuseCPC20PN.H_SelectedChannel].Voltage;
       #H_ETAFuseCPC20PN.H_ChannelInfo.Current := #IO_ETAFuseData.DataCPC20.Fuse[#H_ETAFuseCPC20PN.H_SelectedChannel].Current;
       #H_ETAFuseCPC20PN.H_ChannelInfo.NominalCurrent := #IO_ETAFuseData.DataCPC20.Fuse[#H_ETAFuseCPC20PN.H_SelectedChannel].NominalCurrent;
       #H_ETAFuseCPC20PN.H_ChannelInfo.NominalCurrentConfig := #C_Config.Fuse[#H_ETAFuseCPC20PN.H_SelectedChannel].NominalCurrent;
       #H_ETAFuseCPC20PN.H_ChannelInfo."Name" := #C_Config.Fuse[#H_ETAFuseCPC20PN.H_SelectedChannel]."Name";
       #H_ETAFuseCPC20PN.H_ChannelInfo.Description := #C_Config.Fuse[#H_ETAFuseCPC20PN.H_SelectedChannel].Description;
   END_IF;
   #H_ETAFuseCPC20PN.H_ChannelInfo.Exist := #IO_ETAFuseData.ForHMICPC20.Fuse[#H_ETAFuseCPC20PN.H_SelectedChannel].Used AND #IO_ETAFuseData.ForHMICPC20.Fuse[#H_ETAFuseCPC20PN.H_SelectedChannel].Used;
   #H_ETAFuseCPC20PN."H_SwitchOn/OFFOnlyCabinet" := #IO_ETAFuseData.ForHMICPC20.Fuse[#H_ETAFuseCPC20PN.H_SelectedChannel].Used AND #IO_ETAFuseData.ForHMICPC20.Fuse[#H_ETAFuseCPC20PN.H_SelectedChannel]."SwitchOn/OFFOnlyCabinet";
END_REGION

REGION Network 16: **** 8 - Outputs **** Alarm AB Condition
   // Alarm AB Condition
   #O_AlarmABCondition := "FALSE" OR "FALSE";
   #AlarmABCondition := #O_AlarmABCondition;
END_REGION

REGION Network 17: **** 9 - Alarm Summary **** Alarm A
   // Alarm A
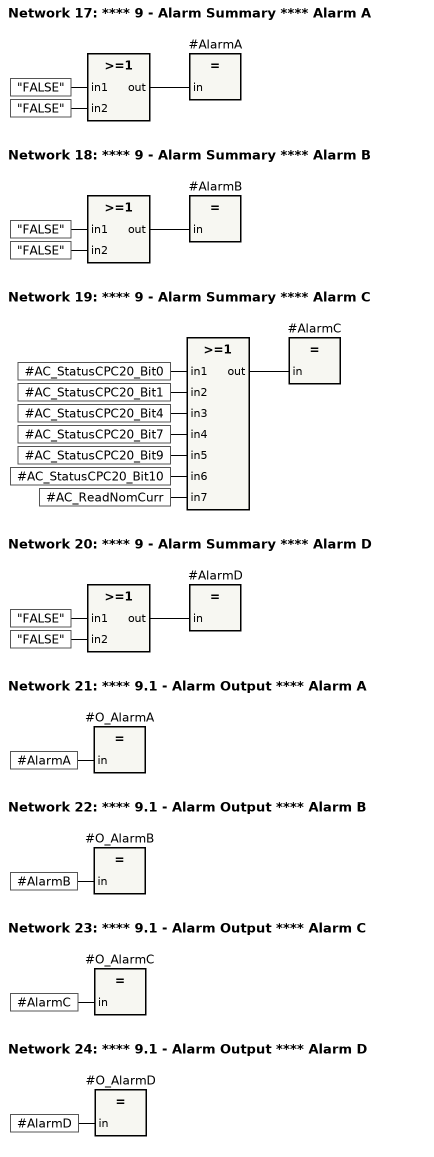
   #AlarmA := "FALSE" OR "FALSE";
END_REGION

REGION Network 18: **** 9 - Alarm Summary **** Alarm B
   // Alarm B
   #AlarmB := "FALSE" OR "FALSE";
END_REGION

REGION Network 19: **** 9 - Alarm Summary **** Alarm C
   // Alarm C
   #AlarmC := #AC_StatusCPC20_Bit0 OR #AC_StatusCPC20_Bit1 OR #AC_StatusCPC20_Bit4 OR #AC_StatusCPC20_Bit7 OR #AC_StatusCPC20_Bit9 OR #AC_StatusCPC20_Bit10 OR #AC_ReadNomCurr;
END_REGION

REGION Network 20: **** 9 - Alarm Summary **** Alarm D
   // Alarm D
   #AlarmD := "FALSE" OR "FALSE";
END_REGION

REGION Network 21: **** 9.1 - Alarm Output **** Alarm A
   // Alarm A
   #O_AlarmA := #AlarmA;
END_REGION

REGION Network 22: **** 9.1 - Alarm Output **** Alarm B
   // Alarm B
   #O_AlarmB := #AlarmB;
END_REGION

REGION Network 23: **** 9.1 - Alarm Output **** Alarm C
   // Alarm C
   #O_AlarmC := #AlarmC;
END_REGION

REGION Network 24: **** 9.1 - Alarm Output **** Alarm D
   // Alarm D
   #O_AlarmD := #AlarmD;
END_REGION

REGION Network 25: **** 9.2 - Alarm DWord**** Alarm To DWord
   // Alarm To Word
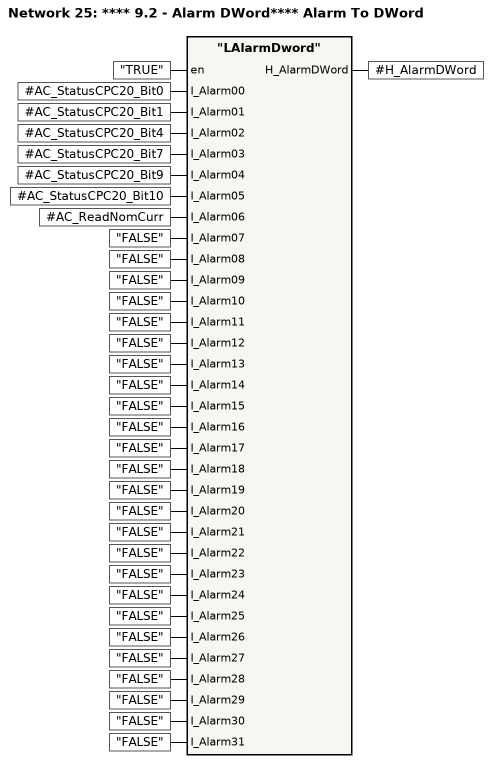
   IF "TRUE" THEN
       "LAlarmDword"(I_Alarm00 := #AC_StatusCPC20_Bit0,
                     I_Alarm01 := #AC_StatusCPC20_Bit1,
                     I_Alarm02 := #AC_StatusCPC20_Bit4,
                     I_Alarm03 := #AC_StatusCPC20_Bit7,
                     I_Alarm04 := #AC_StatusCPC20_Bit9,
                     I_Alarm05 := #AC_StatusCPC20_Bit10,
                     I_Alarm06 := #AC_ReadNomCurr,
                     I_Alarm07 := "FALSE",
                     I_Alarm08 := "FALSE",
                     I_Alarm09 := "FALSE",
                     I_Alarm10 := "FALSE",
                     I_Alarm11 := "FALSE",
                     I_Alarm12 := "FALSE",
                     I_Alarm13 := "FALSE",
                     I_Alarm14 := "FALSE",
                     I_Alarm15 := "FALSE",
                     I_Alarm16 := "FALSE",
                     I_Alarm17 := "FALSE",
                     I_Alarm18 := "FALSE",
                     I_Alarm19 := "FALSE",
                     I_Alarm20 := "FALSE",
                     I_Alarm21 := "FALSE",
                     I_Alarm22 := "FALSE",
                     I_Alarm23 := "FALSE",
                     I_Alarm24 := "FALSE",
                     I_Alarm25 := "FALSE",
                     I_Alarm26 := "FALSE",
                     I_Alarm27 := "FALSE",
                     I_Alarm28 := "FALSE",
                     I_Alarm29 := "FALSE",
                     I_Alarm30 := "FALSE",
                     I_Alarm31 := "FALSE",
                     H_AlarmDWord => #H_AlarmDWord);
   END_IF;
END_REGION
END_FUNCTION_BLOCK

FUNCTION_BLOCK "LETAFuseCPC20PNSub"   // FB1407, SCL
{ S7_Optimized_Access := 'TRUE' }
VERSION : 0.1
// stored: AutoNumber false, IsIECCheckEnabled false, IsRetainMemResEnabled false, MemoryReserve 100, SetENOAutomatically False, UDAEnableTagReadback false
   VAR_INPUT
      I_NewShift { ExternalAccessible := 'False'; ExternalVisible := 'False'; ExternalWritable := 'False'} : Bool;   // NewShift / Morning shift
      I_ReadNomCurr { ExternalAccessible := 'False'; ExternalVisible := 'False'; ExternalWritable := 'False'} : Bool;   // HMI Command - Read nominal current
      I_CancelReadNomCurr { ExternalAccessible := 'False'; ExternalVisible := 'False'; ExternalWritable := 'False'} : Bool;   // HMI Command - Cancel Read nominal current
      C_HWInput { ExternalAccessible := 'False'; ExternalVisible := 'False'; ExternalWritable := 'False'} : HW_IO;   // Slot ID from CPC20PN
      C_Block1_TotalCurrent { ExternalAccessible := 'False'; ExternalVisible := 'False'; ExternalWritable := 'False'} : HW_IO;   // Base Module Slot ID Total Current, 0=not in use.
      C_Block1_StatusControl { ExternalAccessible := 'False'; ExternalVisible := 'False'; ExternalWritable := 'False'} : HW_IO;   // Base Module Slot ID Status / Control, 0=not in use.
      "C_Block1_MeasurementU/I" { ExternalAccessible := 'False'; ExternalVisible := 'False'; ExternalWritable := 'False'} : HW_IO;   // Base Module Slot ID Measurement UI, 0=not in use.
      C_Block2_TotalCurrent { ExternalAccessible := 'False'; ExternalVisible := 'False'; ExternalWritable := 'False'} : HW_IO;   // Extension Module Slot ID Total Current, 0=not in use.
      C_Block2_StatusControl { ExternalAccessible := 'False'; ExternalVisible := 'False'; ExternalWritable := 'False'} : HW_IO;   // Extension Module Slot ID Status / Control, 0=not in use.
      "C_Block2_MeasurementU/I" { ExternalAccessible := 'False'; ExternalVisible := 'False'; ExternalWritable := 'False'} : HW_IO;   // Extension Module Slot ID Measurement UI, 0=not in use.
      C_Config { ExternalAccessible := 'False'; ExternalVisible := 'False'; ExternalWritable := 'False'} : "ETAFuseCPC20PNConfig";   // Config
   END_VAR
   VAR_OUTPUT
      O_StatusCPC20_Bit0 { ExternalAccessible := 'False'; ExternalVisible := 'False'; ExternalWritable := 'False'} : Bool;   // Bit0 = no configuration data available
      O_StatusCPC20_Bit1 { ExternalAccessible := 'False'; ExternalVisible := 'False'; ExternalWritable := 'False'} : Bool;   // Bit1 = invalid configuration data
      O_StatusCPC20_Bit4 { ExternalAccessible := 'False'; ExternalVisible := 'False'; ExternalWritable := 'False'} : Bool;   // Bit4 = command buffer overflow
      O_StatusCPC20_Bit7 { ExternalAccessible := 'False'; ExternalVisible := 'False'; ExternalWritable := 'False'} : Bool;   // Bit7 = no communication with at least one PWR board
      O_StatusCPC20_Bit9 { ExternalAccessible := 'False'; ExternalVisible := 'False'; ExternalWritable := 'False'} : Bool;   // Bit9 = CPC temporary error
      O_StatusCPC20_Bit10 { ExternalAccessible := 'False'; ExternalVisible := 'False'; ExternalWritable := 'False'} : Bool;   // Bit10 = CPC hardware error
      O_ReadNomCurrActive { ExternalAccessible := 'False'; ExternalVisible := 'False'; ExternalWritable := 'False'} : Bool;   // Reading of nominal current is active
      O_ReadNomCurrFuseNr { ExternalAccessible := 'False'; ExternalVisible := 'False'; ExternalWritable := 'False'} : Int;   // Fuse number Reading of nominal current
      O_AlarmReadNomCurr { ExternalAccessible := 'False'; ExternalVisible := 'False'; ExternalWritable := 'False'} : Bool;   // Overtime Reading of nominal current
      O_Block1TotalCurrent { ExternalAccessible := 'False'; ExternalVisible := 'False'; ExternalWritable := 'False'} : Real;   // Total current Block 1
      O_Block2TotalCurrent { ExternalAccessible := 'False'; ExternalVisible := 'False'; ExternalWritable := 'False'} : Real;   // Total current Block 2
   END_VAR
   VAR_IN_OUT
      IO_ETAFuseData : "ETAFuseData";   // ETA fuse status
      H_ETAFuseCPC20PN : "H_ETAFuseCPC20PN";   // Animation
   END_VAR
   VAR
      InitNominalCurrent { ExternalAccessible := 'False'; ExternalVisible := 'False'; ExternalWritable := 'False'} : Bool;   // Read once all Nominal Currents at Startup
      ChannelNumber { ExternalAccessible := 'False'; ExternalVisible := 'False'; ExternalWritable := 'False'} : Int;   // Channel Number
      Block1Size { ExternalAccessible := 'False'; ExternalVisible := 'False'; ExternalWritable := 'False'} : Int;   // Block size
      Block2Size { ExternalAccessible := 'False'; ExternalVisible := 'False'; ExternalWritable := 'False'} : Int;   // Block size
      HardwareID { ExternalAccessible := 'False'; ExternalVisible := 'False'; ExternalWritable := 'False'} : HW_IO;   // HW IO
      i { ExternalAccessible := 'False'; ExternalVisible := 'False'; ExternalWritable := 'False'} : Int;   // Loop Counter
      iCount { ExternalAccessible := 'False'; ExternalVisible := 'False'; ExternalWritable := 'False'} : Int;   // Loop Counter To Go Threw All Channels
      iCalcAddress { ExternalAccessible := 'False'; ExternalVisible := 'False'; ExternalWritable := 'False'} : Int;   // Fuse Adress To Be Calculated
      iCountGet { ExternalAccessible := 'False'; ExternalVisible := 'False'; ExternalWritable := 'False'} : Int;   // Sequence Pointer Get Data
      iCountNominalCurrent { ExternalAccessible := 'False'; ExternalVisible := 'False'; ExternalWritable := 'False'} : Int;   // Loop Counter To Go Threw All Channels
      BuildStatus { ExternalAccessible := 'False'; ExternalVisible := 'False'; ExternalWritable := 'False'} : Word;   // BuildStatus
      iError { ExternalAccessible := 'False'; ExternalVisible := 'False'; ExternalWritable := 'False'} : Int;   // iError
      CalcValue { ExternalAccessible := 'False'; ExternalVisible := 'False'; ExternalWritable := 'False'} : Int;   // CalcValue
      EmptyDataCPC20 { ExternalAccessible := 'False'; ExternalVisible := 'False'; ExternalWritable := 'False'} : Struct   // Empty struct to delete info
         Voltage { ExternalAccessible := 'False'; ExternalVisible := 'False'; ExternalWritable := 'False'} : Real;   // Voltage
         Current { ExternalAccessible := 'False'; ExternalVisible := 'False'; ExternalWritable := 'False'} : Real;   // Current
         NominalCurrent { ExternalAccessible := 'False'; ExternalVisible := 'False'; ExternalWritable := 'False'} : Byte;   // Nominal Current
         Status { ExternalAccessible := 'False'; ExternalVisible := 'False'; ExternalWritable := 'False'} : Byte;   // Status
         Control { ExternalAccessible := 'False'; ExternalVisible := 'False'; ExternalWritable := 'False'} : Byte;   // Control
      END_STRUCT;
      EmptyForHMIFuse { ExternalAccessible := 'False'; ExternalVisible := 'False'; ExternalWritable := 'False'} : Struct   // Empty struct to delete info
         Used { ExternalAccessible := 'False'; ExternalVisible := 'False'; ExternalWritable := 'False'} : Bool;   // Used
         "SwitchOn/OFFOnlyCabinet" { ExternalAccessible := 'False'; ExternalVisible := 'False'; ExternalWritable := 'False'} : Bool;   // Switch On/Off only posible in the cabinet, button on the fuse
         IAnim { ExternalAccessible := 'False'; ExternalVisible := 'False'; ExternalWritable := 'False'} : Word;   // IAnim
         Status { ExternalAccessible := 'False'; ExternalVisible := 'False'; ExternalWritable := 'False'} : Byte;   // Status
         AlarmActive { ExternalAccessible := 'False'; ExternalVisible := 'False'; ExternalWritable := 'False'} : Bool;   // Alarm Active
      END_STRUCT;
      EmptyForHMIChannelInfo { ExternalAccessible := 'False'; ExternalVisible := 'False'; ExternalWritable := 'False'} : Struct   // Empty struct to delete info
         "Name" { ExternalAccessible := 'False'; ExternalVisible := 'False'; ExternalWritable := 'False'} : String[40];   // Fuse name
         Description { ExternalAccessible := 'False'; ExternalVisible := 'False'; ExternalWritable := 'False'} : String[60];   // Description
         Current { ExternalAccessible := 'False'; ExternalVisible := 'False'; ExternalWritable := 'False'} : Real;   // Current
         NominalCurrent { ExternalAccessible := 'False'; ExternalVisible := 'False'; ExternalWritable := 'False'} : Int;   // Nominal Current
      END_STRUCT;
      NonCyclicCommunication { ExternalAccessible := 'False'; ExternalVisible := 'False'; ExternalWritable := 'False'} : Struct   // Non cyclic communication variables
         H_ReadNomCurrTrig { ExternalAccessible := 'False'; ExternalVisible := 'False'; ExternalWritable := 'False'} : Bool;   // HMI button to start reading nominal current
         ReadNomCurrActive { ExternalAccessible := 'False'; ExternalVisible := 'False'; ExternalWritable := 'False'} : Bool;   // Reading of nominal current is active
      END_STRUCT;
      Get { ExternalAccessible := 'False'; ExternalVisible := 'False'; ExternalWritable := 'False'} : Struct   // FB
         bGetData { ExternalAccessible := 'False'; ExternalVisible := 'False'; ExternalWritable := 'False'} : Bool;
         bValid { ExternalAccessible := 'False'; ExternalVisible := 'False'; ExternalWritable := 'False'} : Bool;
         bBusy { ExternalAccessible := 'False'; ExternalVisible := 'False'; ExternalWritable := 'False'} : Bool;
         diIndex { ExternalAccessible := 'False'; ExternalVisible := 'False'; ExternalWritable := 'False'} : DInt;
         uiMlen { ExternalAccessible := 'False'; ExternalVisible := 'False'; ExternalWritable := 'False'} : UInt;
         uilen { ExternalAccessible := 'False'; ExternalVisible := 'False'; ExternalWritable := 'False'} : UInt;
         bError { ExternalAccessible := 'False'; ExternalVisible := 'False'; ExternalWritable := 'False'} : Bool;
         dwState { ExternalAccessible := 'False'; ExternalVisible := 'False'; ExternalWritable := 'False'} : DWord;
         TonError { ExternalAccessible := 'False'; ExternalVisible := 'False'; ExternalWritable := 'False'} : Bool;
         DataByte { ExternalAccessible := 'False'; ExternalVisible := 'False'; ExternalWritable := 'False'} : Array[1..20] of Byte;
      END_STRUCT;
      RDREC_FB { ExternalAccessible := 'False'; ExternalVisible := 'False'; ExternalWritable := 'False'} : RDREC;   // FB
      StatusCPC20 { ExternalAccessible := 'False'; ExternalVisible := 'False'; ExternalWritable := 'False'} : Array[0..1] of Byte;   // Temp
      Current { ExternalAccessible := 'False'; ExternalVisible := 'False'; ExternalWritable := 'False'} : Array[0..1] of Byte;   // Temp
      Status { ExternalAccessible := 'False'; ExternalVisible := 'False'; ExternalWritable := 'False'} : Array[1..32] of Byte;   // Temp
      Control { ExternalAccessible := 'False'; ExternalVisible := 'False'; ExternalWritable := 'False'} : Array[1..32] of Byte;   // Temp
      UI { ExternalAccessible := 'False'; ExternalVisible := 'False'; ExternalWritable := 'False'} : Array[0..130] of Byte;   // Temp
      T_ReadNomCurr { ExternalAccessible := 'False'; ExternalVisible := 'False'; ExternalWritable := 'False'} : TON_TIME;   // Timer
   END_VAR
BEGIN
   (*=================================================================================*)
   (* Init at startup *)
   (*=================================================================================*)
   IF "FirstScan" THEN
       #InitNominalCurrent := True;
   END_IF;

   (*=================================================================================*)
   (* Check number of protectors active *)
   (*=================================================================================*)
   #Block1Size := 0;
   IF #C_Config.Fuse[1].Used THEN
       #Block1Size := 1;
   END_IF;
   IF #C_Config.Fuse[3].Used THEN
       #Block1Size := 2;
   END_IF;
   IF #C_Config.Fuse[5].Used THEN
       #Block1Size := 3;
   END_IF;
   IF #C_Config.Fuse[7].Used THEN
       #Block1Size := 4;
   END_IF;
   IF #C_Config.Fuse[9].Used THEN
       #Block1Size := 5;
   END_IF;
   IF #C_Config.Fuse[11].Used THEN
       #Block1Size := 6;
   END_IF;
   IF #C_Config.Fuse[13].Used THEN
       #Block1Size := 7;
   END_IF;
   IF #C_Config.Fuse[15].Used THEN
       #Block1Size := 8;
   END_IF;
   IF #C_Config.Fuse[17].Used THEN
       #Block1Size := 9;
   END_IF;
   IF #C_Config.Fuse[19].Used THEN
       #Block1Size := 10;
   END_IF;
   IF #C_Config.Fuse[21].Used THEN
       #Block1Size := 11;
   END_IF;
   IF #C_Config.Fuse[23].Used THEN
       #Block1Size := 12;
   END_IF;
   IF #C_Config.Fuse[25].Used THEN
       #Block1Size := 13;
   END_IF;
   IF #C_Config.Fuse[27].Used THEN
       #Block1Size := 14;
   END_IF;
   IF #C_Config.Fuse[29].Used THEN
       #Block1Size := 15;
   END_IF;
   IF #C_Config.Fuse[31].Used THEN
       #Block1Size := 16;
   END_IF;

   #Block2Size := 0;
   IF #C_Config.Fuse[33].Used THEN
       #Block2Size := 1;
   END_IF;
   IF #C_Config.Fuse[35].Used THEN
       #Block2Size :=2;
   END_IF;
   IF #C_Config.Fuse[37].Used THEN
       #Block2Size := 3;
   END_IF;
   IF #C_Config.Fuse[39].Used THEN
       #Block2Size := 4;
   END_IF;
   IF #C_Config.Fuse[41].Used THEN
       #Block2Size := 5;
   END_IF;
   IF #C_Config.Fuse[43].Used THEN
       #Block2Size := 6;
   END_IF;
   IF #C_Config.Fuse[45].Used THEN
       #Block2Size := 7;
   END_IF;
   IF #C_Config.Fuse[47].Used THEN
       #Block2Size := 8;
   END_IF;
   IF #C_Config.Fuse[49].Used THEN
       #Block2Size := 9;
   END_IF;
   IF #C_Config.Fuse[51].Used THEN
       #Block2Size := 10;
   END_IF;
   IF #C_Config.Fuse[53].Used THEN
       #Block2Size := 11;
   END_IF;
   IF #C_Config.Fuse[55].Used THEN
       #Block2Size := 12;
   END_IF;
   IF #C_Config.Fuse[57].Used THEN
       #Block2Size := 13;
   END_IF;
   IF #C_Config.Fuse[59].Used THEN
       #Block2Size := 14;
   END_IF;
   IF #C_Config.Fuse[61].Used THEN
       #Block2Size := 15;
   END_IF;
   IF #C_Config.Fuse[63].Used THEN
       #Block2Size := 16;
   END_IF;

   (*=================================================================================*)
   (* CPC20   ---   Read State *)
   (*=================================================================================*)
   IF #C_HWInput > 0 THEN
       (*Read Data*)
       #iError := DPRD_DAT(LADDR := #C_HWInput, RECORD => #StatusCPC20);
       (*Calculate Value*)
       #BuildStatus := #StatusCPC20[0];
       #BuildStatus := SHL(IN := #BuildStatus, N := 8);
   END_IF;

   #O_StatusCPC20_Bit0 := #BuildStatus.%X0;
   #O_StatusCPC20_Bit1 := #BuildStatus.%X1;
   #O_StatusCPC20_Bit4 := #BuildStatus.%X4;
   #O_StatusCPC20_Bit7 := #BuildStatus.%X7;
   #O_StatusCPC20_Bit9 := #BuildStatus.%X9;
   #O_StatusCPC20_Bit10 := #BuildStatus.%X10;

   (*=================================================================================*)
   (* AM03_1   ---   Read Status + Send Control / Read Voltage + Current *)
   (*=================================================================================*)
   IF #Block1Size > 0 THEN
       // Read Total current and calculate it
       IF #C_Block1_TotalCurrent > 0 THEN
           (*Read Data*)
           #iError := DPRD_DAT(LADDR := #C_Block1_TotalCurrent, RECORD => #Current);
           (*Calculate Value*)
           #CalcValue := #Current[1];
           #CalcValue := SHL(IN := #CalcValue, N := 8);
           #O_Block1TotalCurrent := (#CalcValue + #Current[0]) / 100;
       END_IF;
       (*Status and Control*)
       IF #C_Block1_StatusControl > 0 THEN
           (*Read Inputs*)
           #iError := DPRD_DAT(LADDR := #C_Block1_StatusControl, RECORD => #Status);
           (*Take it over to the Datastructure*)
           FOR #iCount := 1 TO 32 DO
               IF #iCount <= #Block1Size * 2 THEN
                   IF "SimulationActive" THEN
                       "NotUsedBool" := False;
                     ELSE
                       #IO_ETAFuseData.DataCPC20.Fuse[#iCount].Status := #Status[#iCount]; (*Read Status*)
                   END_IF;
                   #Control[#iCount] := #IO_ETAFuseData.DataCPC20.Fuse[#iCount].Control ; (*Write control to the buffer*)
               ELSE
                   #IO_ETAFuseData.DataCPC20.Fuse[#iCount].Status := 255; (*Read Status*)
                   #Control[#iCount] := 0; (*Write control to the buffer*)
               END_IF;
           END_FOR;
           (*Write outputs to the CPC*)
           #iError := DPWR_DAT(LADDR := #C_Block1_StatusControl, RECORD := #Control);
       END_IF;
       (*Measurement preperation*)
       IF #"C_Block1_MeasurementU/I" > 0 THEN
           (*Read measurenets values*)
           #iError := DPRD_DAT(LADDR := #"C_Block1_MeasurementU/I", RECORD => #UI);
           (*Create Measurements*)
           FOR #iCount := 1 TO 32 DO
               (*Calculate new Adress*)
               #iCalcAddress := ((#iCount - 1) * 4);
               IF #iCount <= #Block1Size * 2 THEN
                   (*Calculate current and take it over to the Datastructure*)
                   #CalcValue := #UI[#iCalcAddress + 1]; (*-2*)
                   #CalcValue := SHL(IN := #CalcValue, N := 8);
                   #IO_ETAFuseData.DataCPC20.Fuse[#iCount].Current := INT_TO_REAL(#CalcValue + #UI[#iCalcAddress]) / 100; (*-3*)
                   (*Calculate voltage and take it over to the Datastructure*)
                   #CalcValue := #UI[#iCalcAddress + 3];
                   #CalcValue := SHL(IN := #CalcValue, N := 8); (*-0*)
                   #IO_ETAFuseData.DataCPC20.Fuse[#iCount].Voltage := INT_TO_REAL(#CalcValue + #UI[#iCalcAddress + 2]) / 100; (*-1*)
               ELSE
                   #IO_ETAFuseData.DataCPC20.Fuse[#iCount].Current := 0; (*-3*)
                   #IO_ETAFuseData.DataCPC20.Fuse[#iCount].Voltage := 0; (*-1*)
               END_IF;
           END_FOR;
       END_IF;
   END_IF;

